# B&R Automation Studio project ACOPOStrak (part 2)

#### brdkEMModeToA.c - Converts an equipment module mode constant to a string representation.
```c
#include <brdkEM_func.h>

unsigned long brdkEMModeToA(signed long mode) {
	unsigned long pStr;
	switch(mode) {
		case MODE_UNDEFINED: 	pStr = (unsigned long)&"MODE_UNDEFINED"; 	break;	/* 0 */
		case MODE_PRODUCING: 	pStr = (unsigned long)&"MODE_PRODUCING"; 	break;	/* 1 */
		case MODE_MAINTENANCE: 	pStr = (unsigned long)&"MODE_MAINTENANCE"; 	break;	/* 2 */
		case MODE_MANUAL: 		pStr = (unsigned long)&"MODE_MANUAL"; 		break;	/* 3 */
		case MODE_CLEAN: 		pStr = (unsigned long)&"MODE_CLEAN"; 		break;	/* 16 */
		case MODE_JOG: 			pStr = (unsigned long)&"MODE_JOG"; 			break;	/* 17 */
		case MODE_CIP: 			pStr = (unsigned long)&"MODE_CIP"; 			break;	/* 18 */
		case MODE_CALIBRATING: 	pStr = (unsigned long)&"MODE_CALIBRATING"; 	break;	/* 19 */
		default: break;
	}
	return pStr;
}
```

#### brdkEM_func.c - Internal functions for brdkEM.
```c
#include <brdkEM_func.h>

static unsigned char semCreator = false;
SemCreate_typ SemCreateMUList;
char tmpStr[BRDK_MU_MAX_DESCRIPTION_STRING];

/* initialize the equipment module */
void brdkEMInitialize(brdkEM_typ* this, brdkEM_typ* parent) {
	int i;
	brdk_mu_setup_module_typ module;

	switch(this->internal.initSubstate) {

		case 0:
			if(this->setup.name[0] == 0) ST_name(0,(char*)&this->setup.name,(unsigned char)0); 														/* set module name to task name if not set*/
			brdkStrCpy((unsigned long)this->status.name,(unsigned long)this->setup.name);
			if(this->setup.status.stateSubstateMode) {
				brdkStrCpy((unsigned long)this->status.state,(unsigned long)brdkEMStateToA(this->state));
				brdkStrCpy((unsigned long)this->status.mode,brdkEMModeToA(this->mode));
			}
			if(this->setup.nameIdx > -1) brdkStrAppendUdintToA(this->setup.nameIdx,(unsigned long)&this->status.name, BRDK_STR_CONVERT_DECIMAL,-1);	/* add index to task name */
			this->internal.muList.parentIdx = -1;
			for(i=0; i<= BRDK_EM_MAX_CHILDREN; i++) this->internal.muList.childrenIdx[i] = -1;
			for(i=0; i<= BRDK_MU_MAX_SIBLINGS; i++) this->internal.muList.siblingIdx[i] = -1;
			if(!semCreator) {
				setSubStateText(this,(unsigned long)"creating global semaphore");
				semCreator = true;
				this->internal.initSubstate = 10;
			}
			else this->internal.initSubstate = 20;
			break;

		case 10:
			SemCreateMUList.enable = true;
			SemCreateMUList.initCount = 0;
			SemCreateMUList.maxCount = 1;
			SemCreate(&SemCreateMUList);
			if(SemCreateMUList.status != ERR_OK) setSubStateText(this,(unsigned long)"creating global semaphore");
			else {
				SemRelease(SemCreateMUList.ident);
				this->internal.muList.idx = addToMUList((unsigned long)this,0);
				if(this->internal.muList.idx != -1) {
					emListReady = true;
					this->internal.initSubstate = !this->setup.parent.name[0] ? 40 : 30;	/* check if the module has a parent name assigned */
				}
				else {
					setSubStateText(this,(unsigned long)"em list full. Expand BRDK_EM_MAX_EMS.");
					this->internal.initSubstate = 200;
				}
			}
			break;

		case 20:	/* add module to em list */
			if(!emListReady) setSubStateText(this,(unsigned long)"waiting for em list to be ready");
			else {
				brdkStrCpy((unsigned long)module.name,(unsigned long)this->setup.name);
				module.index = this->setup.nameIdx;
				this->internal.muList.idx = getMUIndex((unsigned long)this, &module);
				if(this->internal.muList.idx != -1) {
					if(moduleSleeping(this->internal.muList.idx)) {
						wakeMU(this->internal.muList.idx,(unsigned long)this);
						if(this->setup.status.last) {
							brdkStrMemMove((unsigned long)this->status.last[1],(unsigned long)this->status.last[0], sizeof(this->status.last[0])*BRDK_MU_MAX_LAST_SIZE);
							brdkStrCpy((unsigned long)this->status.last[0],(unsigned long)"module awake");
						}
						this->internal.initSubstate = 65000;
					}
					else {	/* module name already exists in the list */
						this->status.substate[0] = 0;	/* reset sub state text */
						if(this->setup.status.stateSubstateMode) {
							brdkStrCpy((unsigned long)tmpStr,(unsigned long)"module name ");
							brdkStrCat((unsigned long)tmpStr,(unsigned long)module.name);
							brdkStrCat((unsigned long)tmpStr,(unsigned long)" already used. Rename module.");
							setSubStateText(this,(unsigned long)tmpStr);
						}
						this->internal.muList.idx = -1;
						this->internal.initSubstate = 100;
					}
				}
				else {
					if(SemAcquire(SemCreateMUList.ident) != ERR_OK) setSubStateText(this,(unsigned long)"waiting global semaphore to be free");
					else {
						this->internal.muList.idx = addToMUList((unsigned long)this,0);
						SemRelease(SemCreateMUList.ident);
						setSubStateText(this,(unsigned long)"module added em list");
						if(this->internal.muList.idx != -1) this->internal.initSubstate = !this->setup.parent.name[0] ? 40 : 30;	/* check if the module has a parent name assigned */
						else {
							setSubStateText(this,(unsigned long)"em list full. Expand BRDK_EM_MAX_EMS.");
							this->internal.initSubstate = 200;
						}
					}
				}
			}
			break;

		case 30:	/* find parent */
			this->internal.muList.parentIdx = getMUIndex((unsigned long)this, &this->setup.parent);
			if(this->internal.muList.parentIdx == -1) setSubStateText(this,(unsigned long)"parent not found");
			else this->internal.initSubstate = 40;
			break;

		case 40:	/* find siblings */
			for(i=0; i<= BRDK_MU_MAX_SIBLINGS; i++) {
				if(this->setup.sibling[i].name[0] != 0) {
					this->internal.muList.siblingIdx[i] = getMUIndex((unsigned long)this, &this->setup.sibling[i]);
					if(this->internal.muList.siblingIdx[i] == -1) {
						if(this->setup.status.stateSubstateMode) {
							brdkStrCpy((unsigned long)tmpStr,(unsigned long)"sibling: ");
							brdkStrCat((unsigned long)tmpStr,(unsigned long)this->setup.sibling[i].name);
							brdkStrCat((unsigned long)tmpStr,(unsigned long)" not found");
							setSubStateText(this,(unsigned long)tmpStr);
						}
						break;
					}
				}
			}
			if(i>=BRDK_MU_MAX_SIBLINGS) {
				this->status.substate[0] = 0;	/* reset status text */
				this->internal.initSubstate = this->internal.SemCreate_0.ident == 0 ? 50 : 60;
			}
			break;

		case 50:
			this->internal.SemCreate_0.enable = true;
			this->internal.SemCreate_0.initCount = 0;
			this->internal.SemCreate_0.maxCount = 1;
			SemCreate(&this->internal.SemCreate_0);
			switch(this->internal.SemCreate_0.status) {

				case 0:	/* ERR_OK */
					SemRelease(this->internal.SemCreate_0.ident);		/* release the semaphore so it's ready */
					this->internal.initSubstate = 60;
					break;

				case 65535:	/* ERR_FUB_BUSY */
					break;

				default:
					setSubStateText(this,(unsigned long)"error creating the semaphore");
					break;

			}
			break;

		case 60:
			switch(this->setup.activation) {
				case BRDK_EM_ACTIVATE:
					this->internal.deactivateRequest = false;
					this->internal.initSubstate = 70;
					break;

				case BRDK_EM_ACTIVATE_BY_PARENT:
					if(parent != NULL) {
						if(!parent->internal.deactivateRequest) {
							this->internal.initSubstate = 70;
							this->internal.deactivateRequest = false;
						}
					}
					break;

				default: break;

			}
			break;

		case 70:
			setSubStateText(this,(unsigned long)"register child to parent");
			if(RegisterChild(this, parent) == 0) {
				this->internal.initSubstate = 65000;				/* add child to parent's children list */
				if(this->substate == 0) this->substate = 65000;		/* if substate is still 0 it's auto set to SC */
			}
			break;

		case 100: /* error module name already used. Check if anme is being changed */
			break;

	}
}

/* traverse and find the real interrupter */
unsigned long findInterrupter(unsigned long pEM) {
	if(((brdkEM_typ*)pEM)->internal.pInterrupter != pEM) return findInterrupter(((brdkEM_typ*)pEM)->internal.pInterrupter);
	return pEM;
}

/* flash functionality */
brdk_em_color_typ flashColor(brdkEM_typ* this, brdk_em_color_typ color) {
	if(this->internal.flashTime >= BRDK_EM_FLASH_TIME*2) this->internal.flashTime = 0;
	else this->internal.flashTime += this->status.cycleTime/1000;
	return this->internal.flashTime >= BRDK_EM_FLASH_TIME ? color : WHITE;
}

/* light tree functionality */
void lightTree(brdkEM_typ* this, brdk_em_color_typ color1, brdk_em_color_typ color2) {
	this->status.lightTree.red 		= color1 == RED || color2 == RED;
	this->status.lightTree.yellow 	= color1 == ORANGE || color2 == ORANGE;
	this->status.lightTree.blue 	= color1 == BLUE || color2 == BLUE;
	this->status.lightTree.green 	= color1 == GREEN || color2 == GREEN;
}

/* set default sub state text if not set in program */
void setSubStateText(brdkEM_typ* this, unsigned long pStr) {
	const int MAX_COUNTER = 99999;
	if(this->status.substate[0] == 0 && this->setup.status.stateSubstateMode) {
		if(pStr != 0) {
			brdkStrCpy((unsigned long)this->status.substate,pStr);
			this->internal.statusCnt.internalCounter = this->internal.statusCnt.internalCounter > MAX_COUNTER ? 0 : this->internal.statusCnt.internalCounter+1;		/* increase the status counter to indicate that a change was made */
		}
		else {
			if(this->description[0] == 0) {
				if(this->substate == 0) {
					brdkStrCpy((unsigned long)this->status.substate,(unsigned long)"0: waiting for state change (SC)");
					this->internal.statusCnt.internalCounter = this->internal.statusCnt.internalCounter > MAX_COUNTER ? 0 : this->internal.statusCnt.internalCounter+1;		/* increase the status counter to indicate that a change was made */
				}
				else if(this->internal.cmdSC) {
					switch(this->state) {
						case STATE_DEACTIVATED: brdkStrCpy((unsigned long)this->status.substate, (unsigned long)"SC: waiting for activate command"); break;
						case STATE_STOPPED: case STATE_COMPLETE: brdkStrCpy((unsigned long)this->status.substate, (unsigned long)"SC: waiting for reset command"); break;
						case STATE_IDLE: case STATE_SUSPENDED: case STATE_HELD:	brdkStrCpy((unsigned long)this->status.substate, (unsigned long)"SC: waiting for start command"); break;
						case STATE_ABORTED: brdkStrCpy((unsigned long)this->status.substate, (unsigned long)"SC: waiting for clear command"); break;
						default: brdkStrCpy((unsigned long)this->status.substate, (unsigned long)"SC: waiting for command"); break;
					}
					this->internal.statusCnt.internalCounter = this->internal.statusCnt.internalCounter > MAX_COUNTER ? 0 : this->internal.statusCnt.internalCounter+1;		/* increase the status counter to indicate that a change was made */
				}
			}
			else {
				brdkStrUdintToA(this->substate,(unsigned long)&this->status.substate,BRDK_STR_CONVERT_DECIMAL);
				brdkStrCat((unsigned long)this->status.substate, (unsigned long)": ");
				brdkStrCat((unsigned long)this->status.substate, (unsigned long)this->description);
				this->internal.statusCnt.internalCounter = this->internal.statusCnt.internalCounter > MAX_COUNTER ? 0 : this->internal.statusCnt.internalCounter+1;		/* increase the status counter to indicate that a change was made */
			}
		}
	}
}

/* if the parent mode is changed we also changes it for alle the children */
void setChildrenMode(brdkEM_typ* this) {
	int i;
	for(i=0; i <= BRDK_EM_MAX_CHILDREN; i++) {
		brdkEM_typ* child = getEm(this->internal.muList.childrenIdx[i]);
		if(child != NULL) {
			if(this->setup.reactTo == BRDK_EM_REACT_TO_NONE) child->mode = child->mode;
			else child->mode = this->mode;
		}
		else break;
	}
}

/* CHECKS IF ALL THE CHILDREN IS IN STATE */
void checkChildren(brdkEM_typ* this, brdk_em_states_typ STATE) {
	brdkEM_typ* parent;
	brdkEM_typ* child;
	if(this->internal.cmdSC) {
		int i = 0, j;
		while(i < this->status.childCount) {
			child = getEm(this->internal.muList.childrenIdx[i]);
			if(child != NULL) {
				j = i;
				if(child->state == STATE_ACTIVATING || child->state == STATE_DEACTIVATED || child->state == STATE_DEACTIVATING) i++;
				else {
					switch(child->setup.reactTo) {

						case BRDK_EM_REACT_TO_ALL:
							if(child->state == STATE) i++;
							break;

						case BRDK_EM_REACT_TO_ABORT_AND_STOP:
							if(STATE == STATE_ABORTED || STATE == STATE_STOPPED) {
								if(child->state == STATE) i++;
							}
							else i++;
							break;

						case BRDK_EM_REACT_TO_ABORT_ONLY:
							if(STATE == STATE_ABORTED) {
								if(child->state == STATE) i++;
							}
							else i++;
							break;

						case BRDK_EM_REACT_TO_STOP_ONLY:
							if(STATE == STATE_STOPPED) {
								if(child->state == STATE) i++;
							}
							else i++;
							break;

						case BRDK_EM_REACT_TO_NONE: case BRDK_EM_LISTEN_TO_ABORT_AND_STOP: case BRDK_EM_LISTEN_TO_ABORT_ONLY: case BRDK_EM_LISTEN_TO_STOP_ONLY:
							i++;
							break;

					}
				}
				if(j == i) {	/* index not increased */
					if(child->internal.waitingForIdx != -1) {	/* check to see if a child is also waiting for someone */
						if(this->internal.waitingForIdx != child->internal.waitingForIdx) { /* check if the index has changed - otherwise there is nothing to update in the name */
							if(this->setup.status.waitingFor) brdkStrCpy((unsigned long)this->status.waitingFor.name,(unsigned long)child->status.waitingFor.name);
							this->internal.waitingForIdx = child->internal.waitingForIdx;
						}
						if(this->internal.statusCnt.externalCounter != child->internal.statusCnt.externalCounter) {	/* check if there is a change in the status text */
							if(this->setup.status.waitingFor) brdkStrCpy((unsigned long)this->status.waitingFor.substate,(unsigned long)child->status.waitingFor.substate);
							this->internal.statusCnt.externalCounter = child->internal.statusCnt.externalCounter;
						}
					}
					else {
						if(this->internal.waitingForIdx != child->internal.muList.idx) { /* check if the index has changed - otherwise there is nothing to update in the name */
							if(this->setup.status.stateSubstateMode) {
								brdkStrCpy((unsigned long)this->status.waitingFor.name,(unsigned long)child->setup.name);
								brdkStrCpy((unsigned long)tmpStr, (unsigned long)"SC: waiting for ");
								brdkStrCat((unsigned long)tmpStr, (unsigned long)this->status.waitingFor.name);
								setSubStateText(this,(unsigned long)tmpStr);
							}
							this->internal.waitingForIdx = child->internal.muList.idx;
						}
						if(this->internal.statusCnt.externalCounter != child->internal.statusCnt.internalCounter) {	/* check if there is a change in the status text */
							if(this->setup.status.waitingFor) brdkStrCpy((unsigned long)this->status.waitingFor.substate,(unsigned long)child->status.substate);
							this->internal.statusCnt.externalCounter = child->internal.statusCnt.internalCounter;
						}
					}
					break;
				}
			}
			else break;
		}
		if(parentStateOK(this)) {
			if(i==this->status.childCount) {
				if(this->state == STATE_RESETTING || this->state == STATE_CLEARING) {	/* clear interrupted by data */
					brdkStrMemSet((unsigned long)&this->status.interruptedBy,0,sizeof(this->status.interruptedBy));
					this->internal.pInterrupter = 0;
				}
				if(this->internal.waitingForIdx != -1) {
					if(this->setup.status.waitingFor) brdkStrMemSet((unsigned long)&this->status.waitingFor,0,sizeof(this->status.waitingFor)); /* clear waiting for data */
					this->internal.waitingForIdx = -1;				/* reset waiting for index */
					this->internal.statusCnt.externalCounter = -1;	/* reset external status counter */
				}
				this->state = STATE;
			}
		}
		else {
			if(!this->status.waitingFor.name[0]) {
				parent = getEm(this->internal.muList.parentIdx);
				if(parent != NULL) {
					if(this->internal.waitingForIdx != parent->internal.muList.idx) { /* check if the index has changed - otherwise there is nothing to update */
						this->internal.waitingForIdx = parent->internal.muList.idx;
						if(parent->state == STATE_DEACTIVATED || parent->state == STATE_DEACTIVATING) setSubStateText(this,(unsigned long)"SC: parent is deactivated");
						else setSubStateText(this,(unsigned long)"SC: waiting for parent");
						if(this->setup.status.waitingFor) brdkStrCpy((unsigned long)this->status.waitingFor.name,(unsigned long)parent->setup.name);
					}
					if(this->internal.statusCnt.externalCounter != parent->internal.statusCnt.internalCounter) {	/* check if there is a change in the status text */
						if(this->setup.status.waitingFor) brdkStrCpy((unsigned long)this->status.waitingFor.substate,(unsigned long)parent->status.substate);
						this->internal.statusCnt.externalCounter = parent->internal.statusCnt.internalCounter;
					}
				}
			}
		}
	}
}

/* make sure eventual parent is also in same state before state change */
int parentStateOK(brdkEM_typ* this) {
	int status = false;
	brdkEM_typ* parent = getEm(this->internal.muList.parentIdx);
	if(parent != NULL) {
		switch(this->setup.reactTo) {
			case BRDK_EM_REACT_TO_ALL: 				status = (parent->state == this->state || this->internal.findParent); break;
			case BRDK_EM_REACT_TO_ABORT_AND_STOP: 	status = (this->state == STATE_ABORTING || this->state == STATE_STOPPING) ? (parent->state == this->state) : true; break;
			case BRDK_EM_REACT_TO_ABORT_ONLY:		status = (this->state == STATE_ABORTING) ? (parent->state == this->state) : true; break;
			case BRDK_EM_REACT_TO_STOP_ONLY:		status = (this->state == STATE_STOPPING) ? (parent->state == this->state) : true; break;
			case BRDK_EM_REACT_TO_NONE: case BRDK_EM_LISTEN_TO_ABORT_AND_STOP: case BRDK_EM_LISTEN_TO_ABORT_ONLY: case BRDK_EM_LISTEN_TO_STOP_ONLY:	status = true;
		}
	}
	else status = true;
	return status;
}

/* automatically take the module to it's parents state */
void findParent(brdkEM_typ* this, brdkEM_typ* parent, brdk_em_states_typ cmd, int numArgs, ...) {
	if(parent != NULL) {
		va_list list;
		int i;
		if(this->state == parent->state) this->internal.findParent = false;
		else {
			va_start(list, numArgs);
			for(i=0; i < numArgs; i++) {
				brdk_em_states_typ checkState = va_arg(list, brdk_em_states_typ);
				if(parent->state == checkState) {
					switch(cmd) {
						case STATE_RESETTING: this->cmd.reset = true; break;
						case STATE_STARTING: case STATE_UNHOLDING: case STATE_UNSUSPENDING: this->cmd.start = true; break;
						case STATE_EXECUTE:
							switch(checkState) {
								case STATE_HOLDING: case STATE_HELD: this->cmd.hold = true; break;
								case STATE_SUSPENDING: case STATE_SUSPENDED: this->cmd.suspend = true; break;
								case STATE_COMPLETING: case STATE_COMPLETE: this->cmd.complete = true; break;
								default: break;
							}
							break;
						default: break;
					}
				}
			}
		}
	}
}

/* observes if one of the children is in one of the states */
void observeChildrensState(brdkEM_typ* this, int numArgs, ...) {
	int i,j;
	brdkEM_typ* child;
	va_list list;																					/* define argument list variable */
	for(i=0; i <= BRDK_EM_MAX_CHILDREN; i++) {														/* check all children */
		child = getEm(this->internal.muList.childrenIdx[i]);
		if(child != NULL) {											/* */
			brdk_em_setup_react_typ reactTo = child->setup.reactTo;
			if(reactTo == BRDK_EM_REACT_TO_NONE || reactTo == BRDK_EM_REACT_TO_NONE || reactTo == BRDK_EM_LISTEN_TO_ABORT_AND_STOP || reactTo == BRDK_EM_LISTEN_TO_ABORT_ONLY || reactTo == BRDK_EM_LISTEN_TO_STOP_ONLY) this->state = this->state;
			else {
				va_start(list, numArgs);
				for(j=0; j < numArgs; j++) {
					brdk_em_states_typ child_state = va_arg(list, brdk_em_states_typ);
					if(child->state == child_state) {
						switch(child_state) {

							case STATE_ABORTING:
								if(reactTo == BRDK_EM_REACT_TO_ALL || reactTo == BRDK_EM_REACT_TO_ABORT_AND_STOP || reactTo == BRDK_EM_REACT_TO_ABORT_ONLY) {
									this->internal.pInterrupter = findInterrupter((unsigned long)child); /* save who went in aborted or aborting */
									this->state = STATE_ABORTING;
								}
								break;

							case STATE_STOPPING:
								if((this->internal.cmdSC || this->setup.skipStopSC) && (reactTo == BRDK_EM_REACT_TO_ALL || reactTo == BRDK_EM_REACT_TO_ABORT_AND_STOP || reactTo == BRDK_EM_REACT_TO_STOP_ONLY)) {
									this->internal.pInterrupter = findInterrupter((unsigned long)child); /* save who went in stopped or stopping */
									this->state = STATE_STOPPING;
								}
								break;

							case STATE_SUSPENDING:
								if(this->internal.cmdSC && reactTo == BRDK_EM_REACT_TO_ALL) {
									this->internal.pInterrupter = findInterrupter((unsigned long)child); /* save who went in suspending or suspended */
									this->state = STATE_SUSPENDING;
								}
								break;

							case STATE_HOLDING:
								if(this->internal.cmdSC && reactTo == BRDK_EM_REACT_TO_ALL) {
									this->internal.pInterrupter = findInterrupter((unsigned long)child); /* save who went in holding or held */
									this->state = STATE_HOLDING;
								}
								break;

							default:
								break;

						}
						va_end(list);
						break;
					}
				}
			}
		}
		else {
			va_end(list);
			break;
		}
	}
}

/* observes the parent state by the given states */
void observeParentState(brdkEM_typ* this, brdkEM_typ* parent, int numArgs, ...) {
	int i;
	brdk_em_setup_react_typ reactTo =  this->setup.reactTo;
	if(parent == NULL || reactTo == BRDK_EM_REACT_TO_NONE) this->state = this->state;
	else {
		va_list list;																									/* define argument list variable */
		va_start(list, numArgs);																						/* init list */
		for(i=0; i < numArgs; i++) if(parent->state==va_arg(list, brdk_em_states_typ)) {
			switch(parent->state) {

				case STATE_ABORTING:
					if(reactTo == BRDK_EM_REACT_TO_ALL || reactTo == BRDK_EM_REACT_TO_ABORT_AND_STOP || reactTo == BRDK_EM_REACT_TO_ABORT_ONLY || reactTo == BRDK_EM_LISTEN_TO_ABORT_AND_STOP || reactTo == BRDK_EM_LISTEN_TO_ABORT_ONLY) {
						this->state = parent->state; 	/* get next state item and check if it's equal to parent state. and then set chils state*/
						this->internal.pInterrupter = parent->internal.pInterrupter;
					}
					break;

				case STATE_STOPPING:
					if((this->internal.cmdSC || this->setup.skipStopSC) && (reactTo == BRDK_EM_REACT_TO_ALL || reactTo == BRDK_EM_REACT_TO_ABORT_AND_STOP || reactTo == BRDK_EM_REACT_TO_STOP_ONLY || reactTo == BRDK_EM_LISTEN_TO_STOP_ONLY)) {
						this->state = parent->state; 	/* get next state item and check if it's equal to parent state. and then set chils state*/
						this->internal.pInterrupter = parent->internal.pInterrupter;
					}
					break;

				case STATE_CLEARING:
					if(this->internal.cmdSC && (reactTo == BRDK_EM_REACT_TO_ALL || reactTo == BRDK_EM_REACT_TO_ABORT_AND_STOP || reactTo == BRDK_EM_REACT_TO_ABORT_ONLY)) this->state = parent->state; 	/* get next state item and check if it's equal to parent state. and then set chils state*/
					break;

				default:
					if(this->internal.cmdSC && reactTo == BRDK_EM_REACT_TO_ALL) this->state = parent->state; 	/* get next state item and check if it's equal to parent state. and then set chils state*/
					break;

			}
		}
		va_end(list);
	}																													/* cleanup the system stack */
}

/* check for commands -> STATE_STOPPING means check for command stop... */
void checkCommands(brdkEM_typ* this, brdkEM_typ* parent, int numArgs, ...) {
	brdkEM_typ* child;
	int i,j;
	if(this->internal.cmdSC || this->cmd.abort || (this->cmd.stop && this->setup.skipStopSC)) {
		va_list list;																											/* define argument list variable */
		va_start(list, numArgs);																								/* init list */
		for(i=0; i < numArgs; i++) {
			switch(va_arg(list, brdk_em_states_typ)) {

				case STATE_STOPPING:
					if(this->cmd.stop) {
						i = numArgs;
						this->internal.pInterrupter = (unsigned long)this; /* module interrupted itself */
						this->state = STATE_STOPPING;
					}
					break;

				case STATE_RESETTING:
					if(this->cmd.reset) {
						i = numArgs;
						this->state = STATE_RESETTING;
					}
					break;

				case STATE_CLEARING:
					if(this->cmd.clear) {
						this->state = STATE_CLEARING;
					}
					break;

				case STATE_STARTING:
					if(this->cmd.start) {
						i = numArgs;
						this->state = STATE_STARTING;
					}
					break;

				case STATE_HOLDING:
					if(this->cmd.hold) {
						i = numArgs;
						this->internal.pInterrupter = (unsigned long)this; /* module interrupted itself */
						this->state = STATE_HOLDING;
					}
					break;

				case STATE_UNHOLDING:
					if(this->cmd.start) {
						i = numArgs;
						this->state = STATE_UNHOLDING;
					}
					break;

				case STATE_SUSPENDING:
					if(this->cmd.suspend) {
						i = numArgs;
						this->internal.pInterrupter = (unsigned long)this; /* module interrupted itself */
						this->state = STATE_SUSPENDING;
					}
					break;

				case STATE_UNSUSPENDING:
					if(this->cmd.start) {
						i = numArgs;
						this->state = STATE_UNSUSPENDING;
					}
					break;

				case STATE_COMPLETING:
					if(this->cmd.complete) {
						i = numArgs;
						this->state = STATE_COMPLETING;
					}
					break;

				case STATE_ABORTING:
					if(this->cmd.abort) {
						i = numArgs;
						this->internal.pInterrupter = (unsigned long)this; /* module interrupted itself */
						this->state = STATE_ABORTING;
					}
					break;

				case STATE_ACTIVATING:
					/* wait for initialization complete */
					if(this->internal.initSubstate == 65000) {
						switch(this->setup.activation) {

							case BRDK_EM_ACTIVATE:
								this->state = STATE_ACTIVATING;
								break;

							case BRDK_EM_ACTIVATE_BY_PARENT:
								if(parent != NULL) {
									switch(parent->state) {
										case STATE_DEACTIVATING: case STATE_DEACTIVATED: setSubStateText(this,(unsigned long)"waiting for parent's activation"); break;
										default:
											if(!parent->internal.deactivateRequest) this->state = STATE_ACTIVATING;
											break;
									}
								}
								break;

							default:
								setSubStateText(this, (unsigned long)"waiting for activation");
								break;

						}
					}
					break;

				case STATE_DEACTIVATING:
					switch(this->setup.activation) {

						case BRDK_EM_DEACTIVATE:
							this->internal.deactivateRequest = true;
							for(j=0; j <= BRDK_EM_MAX_CHILDREN; j++) {		/* check all children */
								child = getEm(this->internal.muList.childrenIdx[j]);
								if(child != NULL) {
									if(child->state != STATE_DEACTIVATED && child->state && STATE_DEACTIVATING) break;
								}
							}
							if(j > BRDK_EM_MAX_CHILDREN) {
								i = numArgs;
								this->state = STATE_DEACTIVATING;
							}
							break;

						case BRDK_EM_ACTIVATE_BY_PARENT:
							if(parent != NULL) {
								switch(parent->state) {
									case STATE_DEACTIVATING: case STATE_DEACTIVATED: this->state = STATE_DEACTIVATING; break;

									case STATE_ABORTED: case STATE_STOPPED:
										/* check if parent has deactivation command and then follow */
										if(parent->internal.deactivateRequest) {
											this->internal.deactivateRequest = true;
											for(j=0; j <= BRDK_EM_MAX_CHILDREN; j++) {		/* check all children */
												child = getEm(this->internal.muList.childrenIdx[j]);
												if(child != NULL) {
													if(child->state != STATE_DEACTIVATED && child->state && STATE_DEACTIVATING) break;
												}
											}
											if(j > BRDK_EM_MAX_CHILDREN) {
												i = numArgs;
												this->state = STATE_DEACTIVATING;
											}
										}
										break;

									default: break;
								}
							}
							break;

						default:
							break;

					}
					break;

				default:
					break;

			}
		}
		va_end(list);
		/* check if an unvalid command has been given */
		this->status.unvalidatedCmd = this->state != this->internal.old.state ? false : this->cmd.abort || this->cmd.clear || this->cmd.stop || this->cmd.reset || this->cmd.start || this->cmd.hold || this->cmd.suspend || this->cmd.complete;
	}
}

/* Add's a child to the parents child list */
unsigned short RegisterChild(brdkEM_typ* this, brdkEM_typ* parent) {
	int i=0, j=0;
	if(parent != NULL) {
		for(i=0; i < BRDK_EM_MAX_CHILDREN; i++) {
			if(parent->internal.muList.childrenIdx[i] == this->internal.muList.idx) break;	/* child already exists in array. index is returned */
			else if(parent->internal.muList.childrenIdx[i] == -1) {							/* finds an empty spot in the array */
				j = SemAcquire(parent->internal.SemCreate_0.ident);							/* checks if the semaphore is free */
				if(j == ERR_OK) {
					parent->internal.muList.childrenIdx[i] = this->internal.muList.idx;		/* puts the index in the array */
					parent->status.childCount++;
					SemRelease(parent->internal.SemCreate_0.ident);							/* releases the semaphore again */
					i = ERR_OK;
				}
				else {
					i = j;	/* 33322: Semaphore with the specified ident does not exist   33323: Semaphore is being used */
					if(this->setup.status.stateSubstateMode) {
						brdkStrCpy((unsigned long)tmpStr,(unsigned long)"semaphore error: ");
						brdkStrAppendUdintToA(j,(unsigned long)tmpStr,10,-1);
						setSubStateText(this,(unsigned long)tmpStr);
					}
				}
				break;
			}
		}
		if(i == BRDK_EM_MAX_CHILDREN) {  /* error: child array too small. Solution: make child array bigger */
			setSubStateText(this,(unsigned long)"parent child array full. Increase BRDK_EM_MAX_CHILDREN.");
		}
	}
	return i;
}

/* Unregister a child */
unsigned short UnregisterChild(brdkEM_typ* this, brdkEM_typ* parent) {
	int i=65000,j;
	if(parent != NULL) {
		for(i=0; i < BRDK_EM_MAX_CHILDREN; i++) {
			if(parent->internal.muList.childrenIdx[i] == this->internal.muList.idx) {	/* child found */
				j = SemAcquire(parent->internal.SemCreate_0.ident);	/* checks if the semaphore is free */
				if(j == ERR_OK) {
					parent->internal.muList.childrenIdx[i] = -1;			/* pointer is removed from the array */
					parent->status.childCount--;
					for(j=i; j < BRDK_EM_MAX_CHILDREN; j++) parent->internal.muList.childrenIdx[j] = parent->internal.muList.childrenIdx[j+1];
					SemRelease(parent->internal.SemCreate_0.ident);		/* releases the semaphore again */
					i = ERR_OK;
					this->internal.muList.parentIdx = -1;
				}
				else {
					i = j;	/* 33322: Semaphore with the specified ident does not exist   33323: Semaphore is being used */
					if(this->setup.status.stateSubstateMode) {
						brdkStrCpy((unsigned long)tmpStr,(unsigned long)"semaphore error: ");
						brdkStrAppendUdintToA(j,(unsigned long)tmpStr,10,-1);
						setSubStateText(this,(unsigned long)tmpStr);
					}
				}
				break;
			}
		}
		if(i == BRDK_EM_MAX_CHILDREN) {  /* error: child not found in array */
			setSubStateText(this,(unsigned long)"child not found in parent array.");
		}
	}
	return i;
}
```

#### brdkMU_func.c - Internal functions for brdkMU.
```c
#include <brdkMU_func.h>

enum mu_state_typ
{
	MU_UNVALID,
	MU_ENABLED,
	MU_SLEEPING,
	MU_UPDATING
};

typedef struct brdk_mu_pointers_typ
{	enum mu_state_typ state;
	unsigned char type;	/* 0 = em, 1 = cm */
	unsigned long ptr;
} brdk_mu_pointers_typ;

static brdk_mu_pointers_typ muList[BRDK_MU_MAX_MODULES];
unsigned char emListReady = false;

/* addes a module mu list */
signed long addToMUList(unsigned long this, unsigned char type) {
	signed long i;
	for(i=0; i< BRDK_MU_MAX_MODULES; i++) {
		if(muList[i].ptr == this) return i;	/* module already inside list */
		else if(muList[i].ptr == 0) { 				/* find an empty slot in the list */
			muList[i].ptr = this;
			muList[i].state = MU_ENABLED;
			muList[i].type = type;
			return i;
		}
	}
	return -1;
}

/* returns the index in the em list of the wanted module */
signed long getMUIndex(unsigned long this, brdk_mu_setup_module_typ* module) {
	signed long i;
	brdkEM_typ* em;
	brdkCM_typ* cm;
	for(i=0; i < BRDK_MU_MAX_MODULES; i++) {
		if(muList[i].ptr != this) {
			if(muList[i].ptr != 0){
				if(muList[i].state != MU_UNVALID) {
					switch(muList[i].type) {
						case 0:
							em = (brdkEM_typ*)muList[i].ptr;
							if(!brdkStrCmp((unsigned long)em->setup.name,(unsigned long)module->name) && em->setup.nameIdx == module->index) return i;
							break;

						case 1:
							cm = (brdkCM_typ*)muList[i].ptr;
							if(!brdkStrCmp((unsigned long)cm->setup.name,(unsigned long)module->name) && cm->setup.nameIdx == module->index) return i;
							break;

					}
				}
			}
			else return -1; /* no further modules */
		}
	}
	return -1;
}

/* returns the pointer of the em */
brdkEM_typ* getEm(signed long idx) {
	if(idx != -1) {
		/* TODO - make check of unit type */
		if(muList[idx].state != MU_UNVALID && muList[idx].ptr != 0) return (brdkEM_typ*)muList[idx].ptr;
	}
	return NULL;
}

/* returns the pointer of the em */
brdkCM_typ* getCm(signed long idx) {
	if(idx != -1) {
		/* TODO - make check of unit type */
		if(muList[idx].state != MU_UNVALID && muList[idx].ptr != 0) return (brdkCM_typ*)muList[idx].ptr;
	}
	return NULL;
}

signed long sleepMU(signed long idx, unsigned long this) {
	if(idx != -1) {
		muList[idx].state = MU_UNVALID;
		switch(muList[idx].type) {
			case 0:
				TMP_alloc(sizeof(brdkEM_typ),(void*)&muList[idx].ptr);
				brdkStrMemCpy(muList[idx].ptr,this, sizeof(brdkEM_typ));
				break;

			case 1:
				TMP_alloc(sizeof(brdkCM_typ),(void*)&muList[idx].ptr);
				brdkStrMemCpy(muList[idx].ptr,this, sizeof(brdkCM_typ));
				break;

		}
		muList[idx].state = MU_SLEEPING;
		return idx;
	}
	return -1;
}

signed long wakeMU(signed long idx, unsigned long this) {
	if(idx != -1) {
		if(muList[idx].state == MU_SLEEPING) {
			muList[idx].state = MU_UNVALID;
			switch(muList[idx].type) {
				case 0:
					brdkStrMemCpy(this,muList[idx].ptr, sizeof(brdkEM_typ));	/* UPDATE THIS TO NAME BASE INSTEAD OF MEMORY */
					TMP_free(sizeof(brdkEM_typ),(void*)muList[idx].ptr);
					break;

				case 1:
					brdkStrMemCpy(this,muList[idx].ptr, sizeof(brdkCM_typ));	/* UPDATE THIS TO NAME BASE INSTEAD OF MEMORY */
					TMP_free(sizeof(brdkCM_typ),(void*)muList[idx].ptr);
					break;

			}
			muList[idx].state = MU_ENABLED;
		}
		muList[idx].state = MU_UNVALID;
		muList[idx].ptr = this;
		muList[idx].state = MU_ENABLED;
		return idx;
	}
	return -1;
}

/* returns if a module is sleeping or not */
unsigned char moduleSleeping(signed long idx) {
	return muList[idx].state == MU_SLEEPING;
}

/* updates the siblings state and sub state info for the em function block */
void updateSiblingInfo(signed long (*idxArr)[], brdk_mu_status_module_typ* status) {
	int i;
	brdkEM_typ* sibling;
	for(i=0; i<= BRDK_MU_MAX_SIBLINGS; i++) {
		sibling = getEm((*idxArr)[i]);
		if(sibling != NULL) {
			status[i].state = sibling->state;
			status[i].substate = sibling->substate;
			status[i].sleeping = sibling->status.sleeping;
			status[i].mode = sibling->mode;
		}
	}
}

/* gets the cycle time of the task the em structure is called inside */
unsigned long getCycleTime() {
	RTInfo_typ RTInfo_0;
	RTInfo_0.enable = 1;
	RTInfo(&RTInfo_0);
	return RTInfo_0.cycle_time;
}
```

- CHANGELOG - brdkMU change log file (not shown)

### Library Logical/Libraries/brdkSTR (ANSIC, version 1.04.0) - brdk string handling library. Expands string functionality.

#### brdkSTR.fun
```iecst
FUNCTION brdkStrAppendUdintToA : DINT (*Appends an UDINT to the end of a string. $RETURN=length;Length of the string.*) (*$GROUP=User,$CAT=User,$GROUPICON=User.png,$CATICON=User.png*)
	VAR_INPUT
		value : UDINT; (*UDINT value to be converted.*)
		pString : UDINT; (*String pointer to source string.*)
		base : USINT; (*0,10 = decimal, 2 = binary, 16 = hex.*)
		position : DINT; (*Append position. Negative numbers will count from end of string.*)
	END_VAR
END_FUNCTION

FUNCTION brdkStrAToDint : DINT (*Converts a string to a DINT type. $RETURN=value;DINT value.*) (*$GROUP=User,$CAT=User,$GROUPICON=User.png,$CATICON=User.png*)
	VAR_INPUT
		pString : UDINT; (*String pointer to source string.*)
		base : USINT; (*0,10 = decimal, 2 = binary, 16 = hex.*)
	END_VAR
END_FUNCTION

FUNCTION brdkStrAToUdint : UDINT (*Converts a string to an UDINT type. $RETURN=value;UDINT value.*) (*$GROUP=User,$CAT=User,$GROUPICON=User.png,$CATICON=User.png*)
	VAR_INPUT
		pString : UDINT; (*String pointer to source string.*)
		base : USINT; (*0,10 = decimal, 2 = binary, 16 = hex.*)
	END_VAR
END_FUNCTION

FUNCTION brdkStrCat : UDINT (*Appends a copy of the source string to the end of the destination string. $RETURN=address;Address after the string.*) (*$GROUP=User,$CAT=User,$GROUPICON=User.png,$CATICON=User.png*)
	VAR_INPUT
		pDestination : UDINT; (*Destination string pointer.*)
		pSource : UDINT; (*Source string pointer.*)
	END_VAR
END_FUNCTION

FUNCTION brdkStrCatAtChar : DINT (*Appends a copy of the source string to the char position of the destination string. $RETURN=index;Index in destination string where the source string is appended. -1 if char is not found.*) (*$GROUP=User,$CAT=User,$GROUPICON=User.png,$CATICON=User.png*)
	VAR_INPUT
		pDestination : UDINT; (*Destination string pointer.*)
		pSource : UDINT; (*Source string pointer.*)
		pChar : UDINT; (*Char pointer.*)
		direction : DINT; (*0 = first appearance of char, -1 = last appearance of char.*)
		greedy : BOOL; (*If true the source string is appended to the char position. If false the char is still present in the destination string.*)
	END_VAR
END_FUNCTION

FUNCTION brdkStrCharAt : USINT (*Returns the character at the specified index. $RETURN=coding;ASCII coding of the char.*) (*$GROUP=User,$CAT=User,$GROUPICON=User.png,$CATICON=User.png*)
	VAR_INPUT
		pString : UDINT; (*String pointer to source string.*)
		index : UDINT; (*Look up index.*)
		pChar : UDINT; (*Char pointer to char to look up.*)
	END_VAR
END_FUNCTION

FUNCTION brdkStrCharCount : DINT (*Finds how many times a character appears in a string. $RETURN=count;Char count. -1 if error.*) (*$GROUP=User,$CAT=User,$GROUPICON=User.png,$CATICON=User.png*)
	VAR_INPUT
		pString : UDINT; (*String pointer to source string.*)
		pChar : UDINT; (*Pointer to search char.*)
	END_VAR
END_FUNCTION

FUNCTION brdkStrCmp : DINT (*Compares character(s) from string1 to string2. $RETURN=result;0 means that the two string are equal.*)
	VAR_INPUT
		pString1 : UDINT; (*String1 pointer.*)
		pString2 : UDINT; (*String2 pointer.*)
	END_VAR
END_FUNCTION

FUNCTION brdkStrCpy : UDINT (*Copies a string to another string. $RETURN=address;Address after the string.*) (*$GROUP=User,$CAT=User,$GROUPICON=User.png,$CATICON=User.png*)
	VAR_INPUT
		pDestination : UDINT; (*Destination string pointer.*)
		pSource : UDINT; (*Source string pointer.*)
	END_VAR
END_FUNCTION

FUNCTION brdkStrCrc32 : UDINT (*Calculates a CRC32 checksum based on the input string. $RETURN=checksum;Checksum of the string.*) (*$GROUP=User,$CAT=User,$GROUPICON=User.png,$CATICON=User.png*)
	VAR_INPUT
		pString : UDINT; (*String pointer.*)
	END_VAR
END_FUNCTION

FUNCTION brdkStrDintToA : DINT (*Converts a DINT into a STRING type. $RETURN=length;Length of the string.*) (*$GROUP=User,$CAT=User,$GROUPICON=User.png,$CATICON=User.png*)
	VAR_INPUT
		value : DINT; (*DINT value to be converted.*)
		pString : UDINT; (*String pointer to source string.*)
		base : USINT; (*0,10 = decimal, 2 = binary, 16 = hex.*)
	END_VAR
END_FUNCTION

FUNCTION brdkStrEncode : DINT (*Encodes a string into different formats. $RETURN=address;Address after the string.*) (*$GROUP=User,$CAT=User,$GROUPICON=User.png,$CATICON=User.png*)
	VAR_INPUT
		pDestination : UDINT; (*Destination string pointer.*)
		pSource : UDINT; (*Source string pointer.*)
		format : USINT; (*0 = UTF-8*)
	END_VAR
END_FUNCTION

FUNCTION brdkStrFill : DINT (*Inserts amount of character(s) to the specified position of the string. $RETURN=length;Length of the string. -1 if error.*) (*$GROUP=User,$CAT=User,$GROUPICON=User.png,$CATICON=User.png*)
	VAR_INPUT
		pString : UDINT; (*String pointer to source string.*)
		amount : DINT; (*Fill char amount.*)
		pChar : UDINT; (*Fill char. If 0 whitespace is used.*)
		position : DINT; (*Fill position. Negative numbers will count from end of string.*)
	END_VAR
END_FUNCTION

FUNCTION brdkStrIndexOf : DINT (*Returns the index within this string of the first or last occurrence of the specified character. $RETURN=index;Index of the char. -1 if char is not found.*) (*$GROUP=User,$CAT=User,$GROUPICON=User.png,$CATICON=User.png*)
	VAR_INPUT
		pString : UDINT; (*String pointer to source string.*)
		pChar : UDINT; (*Char pointer to char to look up.*)
		direction : DINT; (*0 = search from left, -1 = search from right.*)
	END_VAR
END_FUNCTION

FUNCTION brdkStrInsertAtPos : DINT (*Inserts a string into another string at a specified position. $RETURN=length;Length of the string. -1 if error.*) (*$GROUP=User,$CAT=User,$GROUPICON=User.png,$CATICON=User.png*)
	VAR_INPUT
		pString : UDINT; (*String pointer to source string.*)
		pInsert : UDINT; (*String pointer to insert string.*)
		position : DINT; (*Insert position. Negative numbers will count from end of string.*)
	END_VAR
END_FUNCTION

FUNCTION brdkStrIsEmpty : BOOL (*Returns false or true depending of characters are present in the first position of the string. $RETURN=false/true;Position [0] = /0 = false. Position [0] != /0 = true.*) (*$GROUP=User,$CAT=User,$GROUPICON=User.png,$CATICON=User.png*)
	VAR_INPUT
		pString : UDINT; (*String pointer.*)
	END_VAR
END_FUNCTION

FUNCTION brdkStrLen : DINT (*Returns the number of characters in a string. Stops at \0. $RETURN=length;length of the string*) (*$GROUP=User,$CAT=User,$GROUPICON=User.png,$CATICON=User.png*)
	VAR_INPUT
		pString : UDINT; (*String pointer.*)
	END_VAR
END_FUNCTION

FUNCTION brdkStrMemCmp : DINT (*Compares amount of character(s) from area1 to area2. $RETURN=result;0 means that the two areas are equal.*) (*$GROUP=User,$CAT=User,$GROUPICON=User.png,$CATICON=User.png*)
	VAR_INPUT
		pArea1 : UDINT; (*Area1 pointer.*)
		pArea2 : UDINT; (*Area2 pointer.*)
		amount : UDINT; (*Amount of character(s) to be comared.*)
	END_VAR
END_FUNCTION

FUNCTION brdkStrMemCpy : UDINT (*Copies amount of character(s) from source to destination. $RETURN=address;Address after the destination.*) (*$GROUP=User,$CAT=User,$GROUPICON=User.png,$CATICON=User.png*)
	VAR_INPUT
		pDestination : UDINT; (*Destination pointer.*)
		pSource : UDINT; (*Source pointer.*)
		amount : UDINT; (*Amount of character(s) to be copied.*)
	END_VAR
END_FUNCTION

FUNCTION brdkStrMemMove : UDINT (*Moves amount of character(s) from source to destination. $RETURN=address;Address after the destination.*) (*$GROUP=User,$CAT=User,$GROUPICON=User.png,$CATICON=User.png*)
	VAR_INPUT
		pDestination : UDINT; (*Destination pointer.*)
		pSource : UDINT; (*Source pointer.*)
		amount : UDINT; (*Amount of character(s) to be moved.*)
	END_VAR
END_FUNCTION

FUNCTION brdkStrMemSet : UDINT (*Fills amount of character(s) to destination. $RETURN=address;Address after the destination.*) (*$GROUP=User,$CAT=User,$GROUPICON=User.png,$CATICON=User.png*)
	VAR_INPUT
		pDestination : UDINT; (*Destination pointer.*)
		value : USINT; (*Initialization value.*)
		amount : UDINT; (*Amount of character(s) to be initialized.*)
	END_VAR
END_FUNCTION

FUNCTION brdkStrMove : UDINT (*Moves a string to another string. $RETURN=address;Address after the string.*) (*$GROUP=User,$CAT=User,$GROUPICON=User.png,$CATICON=User.png*)
	VAR_INPUT
		pDestination : UDINT; (*Destination string pointer.*)
		pSource : UDINT; (*Source string pointer.*)
	END_VAR
END_FUNCTION

FUNCTION brdkStrNCpy : UDINT (*Copies a string to another string. If the function encounters a null character in the source string, the function will add null characters to the destination string until amount character(s) have been written. $RETURN=address;Address after the string.*) (*$GROUP=User,$CAT=User,$GROUPICON=User.png,$CATICON=User.png*)
	VAR_INPUT
		pDestination : UDINT; (*Destination string pointer.*)
		pSource : UDINT; (*Source string pointer.*)
		amount : UDINT; (*Amount of character(s) to be moved.*)
	END_VAR
END_FUNCTION

FUNCTION brdkStrRemove : UDINT (*Removes character(s) from a string from a specified position. $RETURN=address;Address after the string.*) (*$GROUP=User,$CAT=User,$GROUPICON=User.png,$CATICON=User.png*)
	VAR_INPUT
		pString : UDINT; (*Source string pointer.*)
		start : DINT; (*Index of where to start in the string. Negative numbers start from the end of the string.*)
		length : DINT; (*0 means to the end of the string. Negative length is subtracted from the end of the string. Is start is negative length is subtracted from the start of the string. *)
	END_VAR
END_FUNCTION

FUNCTION brdkStrRepeat : DINT (*Repeats a string a specified number of times. $RETURN=length;Length of the string.*) (*$GROUP=User,$CAT=User,$GROUPICON=User.png,$CATICON=User.png*)
	VAR_INPUT
		pString : UDINT; (*String pointer to source string.*)
		times : DINT; (*Number of times the string should be repeated.*)
	END_VAR
END_FUNCTION

FUNCTION brdkStrReplace : DINT (*Replaces some characters with some other characters in a string. $RETURN=number;Number of replacements done.*) (*$GROUP=User,$CAT=User,$GROUPICON=User.png,$CATICON=User.png*)
	VAR_INPUT
		pString : UDINT; (*String pointer to source string.*)
		pFind : UDINT; (*String pointer to find string.*)
		pReplace : UDINT; (*String pointer to replacement string:*)
	END_VAR
END_FUNCTION

FUNCTION brdkStrReverse : DINT (*Reverses a string from start position to end position. $RETURN=count;Number of reverses done. -1 if error.*) (*$GROUP=User,$CAT=User,$GROUPICON=User.png,$CATICON=User.png*)
	VAR_INPUT
		pString : UDINT; (*String pointer to source string.*)
		startPosition : DINT; (*Start position. Must be a positive number and less than length.*)
		endPosition : DINT; (*End position. Must be less than length unless it's a negative numbers which will count from end of string.*)
	END_VAR
END_FUNCTION

FUNCTION brdkStrReverseWords : DINT (*Reverses words in a string. $RETURN=count;Number of words reversed.*) (*$GROUP=User,$CAT=User,$GROUPICON=User.png,$CATICON=User.png*)
	VAR_INPUT
		pString : UDINT; (*String pointer to source string.*)
	END_VAR
END_FUNCTION

FUNCTION brdkStrSearch : DINT (*Searches a string for a specified string. $RETURN=position; Position of the match. -1 if no match.*) (*$GROUP=User,$CAT=User,$GROUPICON=User.png,$CATICON=User.png*)
	VAR_INPUT
		pString : UDINT; (*String pointer to source string.*)
		pSearchString : UDINT; (*String pointer to search string.*)
	END_VAR
END_FUNCTION

FUNCTION brdkStrSlice : DINT (*Slices a part of a string. $RETURN=length;Length of the string. -1 if error.*) (*$GROUP=User,$CAT=User,$GROUPICON=User.png,$CATICON=User.png*)
	VAR_INPUT
		pString : UDINT; (*String pointer to source string.*)
		start : DINT; (*Start position.*)
		end : DINT; (*End position.*)
	END_VAR
END_FUNCTION

FUNCTION brdkStrSubStr : DINT (*Returns a part of a string. $RETURN=length;Length of the destination string. -1 if error.*) (*$GROUP=User,$CAT=User,$GROUPICON=User.png,$CATICON=User.png*)
	VAR_INPUT
		pDestination : UDINT; (*Destination string pointer.*)
		pSource : UDINT; (*Source string pointer.*)
		start : DINT; (*Index of where to start in the string. Negative numbers start from the end of the string.*)
		length : DINT; (*0 means to the end of the string. Negative length is subtracted from the end of the string. Is start is negative length is subtracted from the start of the string. *)
	END_VAR
END_FUNCTION

FUNCTION brdkStrToDec : DINT (*Converts a string of hexadecimal values to ASCII characters. $RETURN=length;Length of the string. -1 if error.*) (*$GROUP=User,$CAT=User,$GROUPICON=User.png,$CATICON=User.png*)
	VAR_INPUT
		pString : UDINT; (*String pointer to source string.*)
	END_VAR
END_FUNCTION

FUNCTION brdkStrToHex : DINT (*Converts a string of ASCII characters to hexadecimal values. $RETURN=length;Length of the string.*) (*$GROUP=User,$CAT=User,$GROUPICON=User.png,$CATICON=User.png*)
	VAR_INPUT
		pString : UDINT; (*String pointer to source string.*)
	END_VAR
END_FUNCTION

FUNCTION brdkStrToLowerCase : DINT (*Converts a string to lowercase letters. $RETURN=number;Number of characters changed.*) (*$GROUP=User,$CAT=User,$GROUPICON=User.png,$CATICON=User.png*)
	VAR_INPUT
		pString : UDINT; (*String pointer to source string.*)
	END_VAR
END_FUNCTION

FUNCTION brdkStrToUpperCase : DINT (*Converts a string to uppercase letters. $RETURN=number;Number of characters changed.*) (*$GROUP=User,$CAT=User,$GROUPICON=User.png,$CATICON=User.png*)
	VAR_INPUT
		pString : UDINT; (*String pointer to source string.*)
	END_VAR
END_FUNCTION

FUNCTION brdkStrToUpperCaseWords : DINT (*Convert the first character of each word to uppercase. (title()). $RETURN=number;Number of characters changed.*) (*$GROUP=User,$CAT=User,$GROUPICON=User.png,$CATICON=User.png*)
	VAR_INPUT
		pString : UDINT; (*String pointer to source string.*)
	END_VAR
END_FUNCTION

FUNCTION brdkStrTrim : DINT (*Removes whitespaces from a string. $RETURN=number;Number of whitespaces removed from string.*) (*$GROUP=User,$CAT=User,$GROUPICON=User.png,$CATICON=User.png*)
	VAR_INPUT
		pString : UDINT; (*String pointer to source string.*)
		direction : DINT; (*0 = both sides, 1 = left side only, -1 = right side only.*)
	END_VAR
END_FUNCTION

FUNCTION brdkStrUdintToA : DINT (*Converts an UDINT into a STRING type. $RETURN=length;Length of the string.*) (*$GROUP=User,$CAT=User,$GROUPICON=User.png,$CATICON=User.png*)
	VAR_INPUT
		value : UDINT; (*UDINT value to be converted.*)
		pString : UDINT; (*String pointer to source string.*)
		base : USINT; (*0,10 = decimal, 2 = binary, 16 = hex.*)
	END_VAR
END_FUNCTION
```

- CHANGELOG - brdkSTR change log (not shown)

### Program Logical/Modules/Main/Main (IEC)

#### Types.typ
```iecst
TYPE
	local_typ : 	STRUCT
		shuttleCount : USINT; (*nr of shuttles added*)
		shuttleFub : ARRAY[0..MAX_NUM_SHUTTLES]OF shuttleFub_typ;
	END_STRUCT;
	shuttleFub_typ : 	STRUCT
		MC_Stop_0 : MC_Stop; (*Function block for stopping shuttles*)
	END_STRUCT;
END_TYPE
```

#### Variables.var
```iecst
VAR
	em : brdkEM; (*Equipment module*)
END_VAR
VAR CONSTANT
	MAX_NUM_SHUTTLES : USINT := 49; (*Maximum Shuttles Handled by the Trak (+1)*)
END_VAR
(*sequence control*)
VAR
	ShuttleAxis : ARRAY[0..MAX_NUM_SHUTTLES] OF McAxisType;
	i : USINT;
END_VAR
(*FUB*)
VAR
	MC_BR_AsmPowerOn_AcpTrak_0 : MC_BR_AsmPowerOn_AcpTrak;
	MC_BR_AsmPowerOff_AcpTrak_0 : MC_BR_AsmPowerOff_AcpTrak;
	MC_BR_AsmGetShuttle_AcpTrak_0 : MC_BR_AsmGetShuttle_AcpTrak;
	this : local_typ;
	MC_BR_AsmReadStatus_AcpTrak_0 : MC_BR_AsmReadStatus_AcpTrak;
	MC_BR_AsmReset_AcpTrak_0 : MC_BR_AsmReset_AcpTrak;
	MC_BR_AsmReadInfo_AcpTrak_0 : MC_BR_AsmReadInfo_AcpTrak;
	SizeofUserdata : UDINT;
	idx : USINT;
	MC_BR_AsmDeleteShuttle_AcpTrak_0 : MC_BR_AsmDeleteShuttle_AcpTrak;
END_VAR
```

#### Main.st
```iecst
PROGRAM _INIT

    (* Write this value into the Size of Userdata in the Shuttle Stereotype configuration *)
    SizeofUserdata := SIZEOF(gShuttleUserData);

	//dummy call
	gTrack1;
	gTrack2;
	gTrack3;
	gTrack4;
	gTrack5;
	gTrack6;

    gMain.status.simulation := DiagCpuIsSimulated();
	IF gMain.status.simulation THEN
		gMain.cmd.reset := TRUE;
	END_IF

END_PROGRAM

PROGRAM _CYCLIC

	IF gMain.status.error THEN
		em.cmd.abort := TRUE;
	END_IF

	CASE em.mode OF

		MODE_PRODUCING:	// #1
			CASE em.state OF

				STATE_STOPPED:

					CASE em.substate OF
						0:
							em.description := 'waiting for communication to segments is ok';
							IF gMain.status.communication THEN
								em.substate := 10;
							END_IF
						10:
							em.description := 'waiting for assembly ready signal - estop ok?';
							IF gMain.status.ready OR gMain.status.power THEN
								em.substate := 20;
							ELSIF NOT gMain.status.communication THEN
								em.substate := 0;
							END_IF
						20:
							em.description := 'track ready, waiting for reset cmd';
							IF gMain.cmd.reset THEN
								gMain.cmd.reset := FALSE;
								idx := this.shuttleCount := 0;
								em.cmd.reset	:= TRUE;
								em.cmd.sc 		:= TRUE;
							ELSIF NOT gMain.status.ready OR NOT gMain.status.communication THEN
								gMain.cmd.reset := FALSE;
								em.cmd.sc 		:= FALSE;
								em.substate := 0;
							END_IF
					END_CASE

				STATE_RESETTING:

					CASE em.substate OF
						0:
							em.description := 'power on';
							IF MC_BR_AsmReadStatus_AcpTrak_0.AssemblyReady AND MC_BR_AsmReadStatus_AcpTrak_0.Valid THEN
								MC_BR_AsmPowerOn_AcpTrak_0.Execute 	:= FALSE;
								em.substate							:= 10;
							ELSE
								MC_BR_AsmPowerOn_AcpTrak_0.Execute := TRUE;
							END_IF
						10:
							em.description := 'check for shuttles on this sector';
							MC_BR_AsmGetShuttle_AcpTrak_0.Enable := TRUE;
							IF MC_BR_AsmGetShuttle_AcpTrak_0.Valid THEN
								idx := 0;
								em.substate := 20;
							END_IF
						20:
							em.description := 'loop through shuttles and save it';
							MC_BR_AsmGetShuttle_AcpTrak_0.Next := FALSE;
							IF MC_BR_AsmGetShuttle_AcpTrak_0.TotalCount > 0 THEN
								ShuttleAxis[idx] := MC_BR_AsmGetShuttle_AcpTrak_0.Axis;
								em.substate := 30;
							END_IF
						30:
							em.description := 'get next shuttle or move on';
							IF MC_BR_AsmGetShuttle_AcpTrak_0.RemainingCount > 0 THEN
								MC_BR_AsmGetShuttle_AcpTrak_0.Next := TRUE;
								idx := idx + 1;
								em.substate := 20;
							ELSE
								em.substate := SC;
							END_IF
						SC://state complete
							em.description := 'waiting for childs';
							this.shuttleCount := idx;
							idx := 0;
							MC_BR_AsmGetShuttle_AcpTrak_0.Enable := FALSE;
							em.cmd.sc := TRUE;
					END_CASE

				STATE_IDLE:
					em.description := 'Wait for start command';
					IF gMain.cmd.start THEN
						gMain.cmd.start := FALSE;
						em.cmd.start	:= TRUE;
						em.cmd.sc		:= TRUE;
					END_IF

				STATE_STARTING:
					em.cmd.sc := TRUE;
					em.description := 'waiting for children';

				STATE_EXECUTE:
					em.description := 'Waiting for stop command';
					IF gMain.cmd.stop THEN
						gMain.cmd.stop 	:= FALSE;
						em.cmd.stop 	:= TRUE;
					END_IF
					em.cmd.sc := TRUE;

				STATE_STOPPING:
					em.description := 'Stop all shuttles - normal';
					FOR i := 0 TO MAX_NUM_SHUTTLES DO
						this.shuttleFub[i].MC_Stop_0.Deceleration := 10.0;
						this.shuttleFub[i].MC_Stop_0.Execute := TRUE;
					END_FOR
					em.cmd.sc := TRUE;

				STATE_ABORTING:
					em.description := 'Stop all shuttles - fast';
					FOR i := 0 TO MAX_NUM_SHUTTLES DO
						this.shuttleFub[i].MC_Stop_0.Deceleration := 35.0;
						this.shuttleFub[i].MC_Stop_0.Execute := TRUE;
					END_FOR
					em.cmd.sc := TRUE;

				STATE_ABORTED:
					em.description := 'assembly fault';
					IF gMain.cmd.clear THEN
						gMain.cmd.clear := FALSE;
						em.cmd.clear := TRUE;
					END_IF

				STATE_CLEARING:
					CASE em.substate OF
						0:
							em.description := 'delete all shuttles';
							MC_BR_AsmDeleteShuttle_AcpTrak_0.Execute := TRUE;
							MC_BR_AsmDeleteShuttle_AcpTrak_0.Command :=  mcACPTRAK_SH_DELETE_ALL;
							em.substate := 10;

						10:
							em.description := 'waiting for delete all shuttles done';
							IF MC_BR_AsmDeleteShuttle_AcpTrak_0.Done THEN
								MC_BR_AsmDeleteShuttle_AcpTrak_0.Execute := FALSE;
								em.substate := 20;
							END_IF

						20:
							em.description := 'reset error';
							brsmemset(ADR(ShuttleAxis),0,SIZEOF(ShuttleAxis));
							MC_BR_AsmReset_AcpTrak_0.Execute := TRUE;
							em.substate := 30;

						30:
							em.description := 'waiting for error reset done';
							IF MC_BR_AsmReset_AcpTrak_0.Done OR NOT gMain.status.error THEN
								MC_BR_AsmReset_AcpTrak_0.Execute := FALSE;
								em.cmd.sc := TRUE;
							END_IF
					END_CASE

				ELSE	// if need add the missing states
					em.cmd.sc := TRUE;

			END_CASE

		MODE_MANUAL: // #3
			CASE em.state OF

				STATE_STOPPED:
					em.description := 'this is a good place to write what the module is waiting for';

				STATE_RESETTING:

				STATE_IDLE:

				STATE_STARTING:

				STATE_EXECUTE:

				STATE_STOPPING:

				ELSE	// if need add the missing states
					em.cmd.sc := TRUE;

			END_CASE

		ELSE
			em.cmd.sc := TRUE;

	END_CASE

	FOR i := 0 TO MAX_NUM_SHUTTLES DO
		IF ShuttleAxis[i].controlif <> 0 THEN
			this.shuttleFub[i].MC_Stop_0.Axis			:= ADR(ShuttleAxis[i]);
			this.shuttleFub[i].MC_Stop_0.Deceleration	:= 2.0;
			this.shuttleFub[i].MC_Stop_0();
			IF this.shuttleFub[i].MC_Stop_0.Done THEN
				this.shuttleFub[i].MC_Stop_0.Execute := FALSE;
			END_IF
		ELSE
			this.shuttleFub[i].MC_Stop_0.Execute := FALSE;
		END_IF
	END_FOR

	MC_BR_AsmPowerOn_AcpTrak_0.Assembly := ADR(gAssembly_1);
	MC_BR_AsmPowerOn_AcpTrak_0();

	MC_BR_AsmPowerOff_AcpTrak_0.Assembly := ADR(gAssembly_1);
	MC_BR_AsmPowerOff_AcpTrak_0();

	MC_BR_AsmReadStatus_AcpTrak_0.Assembly 	:= ADR(gAssembly_1);
	MC_BR_AsmReadStatus_AcpTrak_0.Enable	:= TRUE;
	MC_BR_AsmReadStatus_AcpTrak_0();

	MC_BR_AsmGetShuttle_AcpTrak_0.Assembly	:= ADR(gAssembly_1);
	MC_BR_AsmGetShuttle_AcpTrak_0();

	MC_BR_AsmReadInfo_AcpTrak_0.Assembly := ADR(gAssembly_1);
	MC_BR_AsmReadInfo_AcpTrak_0.Enable := TRUE;
	MC_BR_AsmReadInfo_AcpTrak_0();

	MC_BR_AsmReset_AcpTrak_0.Assembly := ADR(gAssembly_1);
	MC_BR_AsmReset_AcpTrak_0();

	MC_BR_AsmDeleteShuttle_AcpTrak_0.Assembly := ADR(gAssembly_1);
	MC_BR_AsmDeleteShuttle_AcpTrak_0();

	em();								// call the module

	gMain.status.ready := MC_BR_AsmReadInfo_AcpTrak_0.AssemblyInfo.ReadyForPowerOn AND MC_BR_AsmReadInfo_AcpTrak_0.Valid;
	gMain.status.power := MC_BR_AsmReadStatus_AcpTrak_0.AssemblyReady AND MC_BR_AsmReadStatus_AcpTrak_0.Valid;
	gMain.status.communication := MC_BR_AsmReadInfo_AcpTrak_0.AssemblyInfo.CommunicationReady AND MC_BR_AsmReadInfo_AcpTrak_0.Valid;
	gMain.status.error := MC_BR_AsmReadStatus_AcpTrak_0.AssemblyErrorStop AND MC_BR_AsmReadStatus_AcpTrak_0.Valid;

END_PROGRAM

PROGRAM _EXIT
	(* Insert code here *)

END_PROGRAM
```

### MainGlobal.typ - Global data types
```iecst
TYPE
	main_interface_typ : 	STRUCT
		cmd : main_if_cmd_typ;
		status : main_if_status_typ;
	END_STRUCT;
	main_if_cmd_typ : 	STRUCT
		reset : BOOL; (*Power on assembly*)
		start : BOOL; (*Start all shuttles*)
		stop : BOOL; (*Stop all shuttles*)
		clear : BOOL; (*Clear assembly error*)
		safety : main_if_cmd_safety_typ; (*safety*)
	END_STRUCT;
	main_if_cmd_safety_typ : 	STRUCT
		reset : BOOL; (*reset safety*)
	END_STRUCT;
	main_if_status_typ : 	STRUCT
		power : BOOL; (*power on*)
		ready : BOOL; (*ready to power on*)
		error : BOOL; (*assembly fault*)
		simulation : BOOL; (*target is simulated*)
		communication : BOOL; (*communication to all segments ok*)
		safety : main_if_status_safety_typ; (*safety*)
	END_STRUCT;
	main_if_status_safety_typ : 	STRUCT
		moduleOK : BOOL; (*communication ok*)
		ready : BOOL; (*safety ready*)
		resetNeeded : BOOL; (*safety reset needed*)
		started : BOOL; (*safety running*)
	END_STRUCT;
END_TYPE
```

### MainGlobal.var - Global variables
```iecst
VAR
	gMain : main_interface_typ;
END_VAR
```

### Program Logical/Modules/Sectors/Track1Sector/Track1Sector (IEC) - Task for handling Track 2 sectors

#### Main.st - Init, cyclic, exit code
```iecst
PROGRAM _INIT

	MC_BR_TrgPointEnable_AcpTrak_0.Enable := TRUE;
	MC_BR_BarrierCommand_AcpTrak_0.Command := mcACPTRAK_BARRIER_ADD_TICKETS;
	MC_BR_BarrierCommand_AcpTrak_0.AdvancedParameters.TicketCount := 1;

	myTestDirection := mcDIR_POSITIVE;

END_PROGRAM

PROGRAM _CYCLIC

	em.setup.parent.name := 'Main';

	setup;

	CASE em.state OF
		STATE_STOPPED:
			idx := 0;
			MC_BR_SecGetShuttle_AcpTrak_0.Enable := FALSE;
			em.cmd.sc := TRUE;

		STATE_RESETTING:
			CASE em.substate OF
				0:
					em.description := 'check for shuttles on this sector';
					MC_BR_SecGetShuttle_AcpTrak_0.Enable := gMain.status.power;
					IF MC_BR_SecGetShuttle_AcpTrak_0.Valid THEN
						em.substate := 10;
					END_IF
				10:
					em.description := 'loop through shuttles and save it';
					MC_BR_SecGetShuttle_AcpTrak_0.Next := FALSE;
					IF MC_BR_SecGetShuttle_AcpTrak_0.TotalCount > 0 THEN
						this.axis[idx] := MC_BR_SecGetShuttle_AcpTrak_0.Axis;
						em.substate := 20;
					ELSE
						em.cmd.sc := TRUE; //no shuttles
					END_IF
				20:
					em.description := 'get next shuttle or move on';
					IF MC_BR_SecGetShuttle_AcpTrak_0.RemainingCount > 0 THEN
						MC_BR_SecGetShuttle_AcpTrak_0.Next := TRUE;
						idx := idx + 1;
						em.substate := 10;
					ELSE
						idx := 0;
						em.cmd.sc := TRUE;
					END_IF
			END_CASE

		STATE_STARTING:
			CASE em.substate OF
				0:
					em.description := 'start shuttle movement';
					IF MC_BR_SecGetShuttle_AcpTrak_0.TotalCount > 0 THEN
						MC_BR_ElasticMoveVel_AcpTrak_0.Axis 	:= ADR(this.axis[idx]);
						MC_BR_ElasticMoveVel_AcpTrak_0.Execute 	:= TRUE;
						em.substate := 10;
					ELSE
						em.cmd.sc := TRUE; // no shuttles
					END_IF
				10:
					em.description := 'need a scan before checking if the fub is active or in velocity'; //when changing axis (still active from last execute)
					IF MC_BR_ElasticMoveVel_AcpTrak_0.Active THEN
						MC_BR_ElasticMoveVel_AcpTrak_0.Execute := FALSE;
						idx := idx+1;
						em.substate := 20;
					ELSIF MC_BR_ElasticMoveVel_AcpTrak_0.Error THEN
						//todo: error handling
					END_IF
				20:
					em.description := 'move on or next shuttle';
					IF MC_BR_SecGetShuttle_AcpTrak_0.TotalCount = idx THEN
						idx := 0; 	//done
						em.cmd.sc := TRUE;
					ELSE			//next
						em.substate := 0;
					END_IF
			END_CASE

		STATE_EXECUTE:
			em.cmd.sc := TRUE;
			CASE em.substate OF
				0:
					em.description := 'waiting for shuttle';
					IF MC_BR_TrgPointEnable_AcpTrak_0.EventCount > 0 AND MC_BR_TrgPointEnable_AcpTrak_0.Valid THEN
						em.substate := 10;
					END_IF
				10:
					em.description := 'get axis id';
					MC_BR_TrgPointGetInfo_AcpTrak_0.Execute := TRUE;
					IF MC_BR_TrgPointGetInfo_AcpTrak_0.Done THEN
						axis := MC_BR_TrgPointGetInfo_AcpTrak_0.TrgPointInfo.Axis;
						MC_BR_TrgPointGetInfo_AcpTrak_0.Execute := FALSE;
						em.substate := 20;
					END_IF
				20:
					em.description := 'read axis user data';
					MC_BR_ShCopyUserData_AcpTrak_0.Axis 		:= ADR(axis);    				//Zuweisen der Achsreferenz
		            MC_BR_ShCopyUserData_AcpTrak_0.DataAddress 	:= ADR(this.userData);          //Zuweisen der zu lesenden Prozessvariable
		            MC_BR_ShCopyUserData_AcpTrak_0.DataSize 	:= SIZEOF(this.userData);       //Zuweisen der Länge der Prozessvariable
		            MC_BR_ShCopyUserData_AcpTrak_0.Mode 		:= mcACPTRAK_USERDATA_GET;      //Modus auf Schreiben setzen
		            MC_BR_ShCopyUserData_AcpTrak_0.Execute 		:= TRUE;                        //Werte der Prozessvariable auf die Anwenderdaten des Shuttles kopieren
		            IF MC_BR_ShCopyUserData_AcpTrak_0.Done THEN                            		//Kopieren der Werte war erfolgreich
		                MC_BR_ShCopyUserData_AcpTrak_0.Execute := FALSE;
		                em.substate := 30;
		            END_IF
		        30:
					em.description := 'write axis user data';
					MC_BR_ShCopyUserData_AcpTrak_0.Axis 		:= ADR(axis);    				 //Zuweisen der Achsreferenz
					MC_BR_ShCopyUserData_AcpTrak_0.DataAddress 	:= ADR(this.userData);           //Zuweisen der zu beschreibenden Prozessvariable
		            MC_BR_ShCopyUserData_AcpTrak_0.DataSize 	:= SIZEOF(this.userData);        //Zuweisen der Länge der Prozessvariable
		            MC_BR_ShCopyUserData_AcpTrak_0.Mode 		:= mcACPTRAK_USERDATA_SET;       //Modus auf Lesen setzen
		            MC_BR_ShCopyUserData_AcpTrak_0.Execute 		:= TRUE;                         //Werte der Anwenderdaten des Shuttles auf die Prozessvariable kopieren
		            IF MC_BR_ShCopyUserData_AcpTrak_0.Done THEN                            		 //Kopieren der Werte war erfolgreich
		                MC_BR_ShCopyUserData_AcpTrak_0.Execute := FALSE;
		                em.substate := 40;
		            END_IF
				40:
					em.description := 'send shuttle to next sector';
					MC_BR_RoutedMoveVel_AcpTrak_0.Axis 		:= ADR(axis);
					MC_BR_RoutedMoveVel_AcpTrak_0.Execute 	:= TRUE;
					em.substate := 50;
				50:
					em.description := 'need a scan before checking if the fub is active'; //when changing axis
					IF MC_BR_RoutedMoveVel_AcpTrak_0.Active THEN
						MC_BR_RoutedMoveVel_AcpTrak_0.Execute := FALSE;
						em.substate := 0;
					END_IF
			END_CASE

			STATE_CLEARING:
				brsmemset(ADR(this.axis),0,SIZEOF(this.axis));
				em.cmd.sc := TRUE;
	ELSE
		em.cmd.sc := TRUE;
	END_CASE

	em();

	MC_BR_SecGetShuttle_AcpTrak_0();
	MC_BR_TrgPointEnable_AcpTrak_0();
	MC_BR_TrgPointGetInfo_AcpTrak_0();
	MC_BR_RoutedMoveVel_AcpTrak_0();
	MC_BR_ElasticMoveVel_AcpTrak_0();
	MC_BR_ShCopyUserData_AcpTrak_0();
	MC_BR_BarrierCommand_AcpTrak_0();
	IF MC_BR_BarrierCommand_AcpTrak_0.Done THEN
		MC_BR_BarrierCommand_AcpTrak_0.Execute := FALSE;
	END_IF

	MC_BR_BarrierReadInfo_AcpTrak_0(Enable := TRUE);

END_PROGRAM

PROGRAM _EXIT
	(* Insert code here *)

END_PROGRAM
```

#### setup.st
```iecst
ACTION setup:

	gTrack1.velocity     := SEL(gTrack1.velocity <> 0.0, 0.5, gTrack1.velocity); //default 0.5
    gTrack1.acceleration := SEL(gTrack1.acceleration <> 0.0, 1.0, gTrack1.acceleration); //default 1.0
    gTrack1.deceleration := SEL(gTrack1.deceleration <> 0.0, 1.0, gTrack1.deceleration); //default 1.0

	MC_BR_SecGetShuttle_AcpTrak_0.Sector := ADR(SectorTrack1);	//current sector

	MC_BR_TrgPointEnable_AcpTrak_0.Enable := FALSE; //<--- only valid for Track1 (not used)
	MC_BR_TrgPointEnable_AcpTrak_0.ProcessPoint := ADR(PP_Track1);
	MC_BR_TrgPointGetInfo_AcpTrak_0.ProcessPoint := ADR(PP_Track1);

	MC_BR_RoutedMoveVel_AcpTrak_0.Sector 	:= ADR(SectorTrack4); //next sector
	MC_BR_RoutedMoveVel_AcpTrak_0.Position 	:= 0.0;
	MC_BR_RoutedMoveVel_AcpTrak_0.AdvancedParameters.StartDirection 	:= mcDIR_UNDEFINED;
	MC_BR_RoutedMoveVel_AcpTrak_0.AdvancedParameters.EndDirection 		:= mcDIR_UNDEFINED;
	MC_BR_RoutedMoveVel_AcpTrak_0.AdvancedParameters.ShuttleOrientation := mcDIR_UNDEFINED;
	MC_BR_RoutedMoveVel_AcpTrak_0.Velocity 		:= gTrack1.velocity;
	MC_BR_RoutedMoveVel_AcpTrak_0.RouteVelocity := gTrack1.velocity;
	MC_BR_RoutedMoveVel_AcpTrak_0.Acceleration 	:= gTrack1.acceleration;
	MC_BR_RoutedMoveVel_AcpTrak_0.Deceleration 	:= gTrack1.deceleration;

	MC_BR_ElasticMoveVel_AcpTrak_0.Acceleration := gTrack1.acceleration;
	MC_BR_ElasticMoveVel_AcpTrak_0.Deceleration := gTrack1.deceleration;
	MC_BR_ElasticMoveVel_AcpTrak_0.Velocity 	:= gTrack1.velocity;
	MC_BR_ElasticMoveVel_AcpTrak_0.Direction 	:= myTestDirection;

	MC_BR_BarrierCommand_AcpTrak_0.ProcessPoint := ADR(PP_Track1);
	MC_BR_BarrierReadInfo_AcpTrak_0.ProcessPoint := ADR(PP_Track1);

	this.userData.Color := SHUTTLE_COLOR_BLUE;

END_ACTION
```

#### Variables.var - Local variables
```iecst
VAR
	idx : USINT;
	em : brdkEM; (*Equipment module*)
	this : this_typ;
	MC_BR_TrgPointEnable_AcpTrak_0 : MC_BR_TrgPointEnable_AcpTrak;
	MC_BR_TrgPointGetInfo_AcpTrak_0 : MC_BR_TrgPointGetInfo_AcpTrak;
	MC_BR_RoutedMoveVel_AcpTrak_0 : MC_BR_RoutedMoveVel_AcpTrak;
	MC_BR_SecGetShuttle_AcpTrak_0 : MC_BR_SecGetShuttle_AcpTrak;
	MC_BR_ElasticMoveVel_AcpTrak_0 : MC_BR_ElasticMoveVel_AcpTrak;
	axis : McAxisType;
	MC_BR_ShCopyUserData_AcpTrak_0 : MC_BR_ShCopyUserData_AcpTrak;
	MC_BR_BarrierCommand_AcpTrak_0 : MC_BR_BarrierCommand_AcpTrak;
END_VAR
(*Insert your comment here.*)
VAR
	cm : brdkCM;
	MC_BR_TrgPointEnable_PreTrak : MC_BR_TrgPointEnable_AcpTrak;
	MC_BR_TrgPointGetInfo_PreTrak : MC_BR_TrgPointGetInfo_AcpTrak;
	MC_BR_RoutedMoveVel_PreTrak : MC_BR_RoutedMoveVel_AcpTrak;
	MC_BR_BarrierReadInfo_AcpTrak_0 : MC_BR_BarrierReadInfo_AcpTrak;
	myTestDirection : McDirectionEnum;
END_VAR
```

#### Types.typ - Local data types
```iecst
TYPE
	this_typ : 	STRUCT
		axis : ARRAY[0..29]OF McAxisType;
		shiftSector : BOOL;
		userData : ShuttleUserData_typ;
		selector : trak_parameter_selector_typ;
		preAxis : McAxisType;
		counter : USINT;
	END_STRUCT;
END_TYPE
```

### Track1Global.typ - Global data types
```iecst
TYPE
	trak_parameter_typ : 	STRUCT
		velocity : REAL;
		acceleration : REAL;
		deceleration : REAL;
		selector : trak_parameter_selector_typ;
	END_STRUCT;
	trak_parameter_selector_typ :
		(
		TRAK_SELECTOR_ALL := 0,
		TRAK_SELECTOR_NONE := 1,
		TRAK_SELECTOR_2ND := 2,
		TRAK_SELECTOR_3RD := 3,
		TRAK_SELECTOR_4TH := 4
		);
END_TYPE
```

### Track1Global.var - Global variables
```iecst
VAR RETAIN
	gTrack1 : trak_parameter_typ;
END_VAR
```

### Program Logical/Modules/Sectors/Track2Sector/Track2Sector (IEC) - Task for handling Track 2 sectors

- Main.st (reference to Logical/Modules/Sectors/Track1Sector/Track1Sector/Main.st)

#### setup.st
```iecst
ACTION setup:

	gTrack2.velocity     := SEL(gTrack2.velocity <> 0.0, 0.5, gTrack2.velocity); //default 0.5
    gTrack2.acceleration := SEL(gTrack2.acceleration <> 0.0, 1.0, gTrack2.acceleration); //default 1.0
    gTrack2.deceleration := SEL(gTrack2.deceleration <> 0.0, 1.0, gTrack2.deceleration); //default 1.0

	MC_BR_SecGetShuttle_AcpTrak_0.Sector := ADR(SectorTrack2);	//current sector

	MC_BR_TrgPointEnable_AcpTrak_0.ProcessPoint := ADR(PP_Track2);
	MC_BR_TrgPointGetInfo_AcpTrak_0.ProcessPoint := ADR(PP_Track2);

	MC_BR_RoutedMoveVel_AcpTrak_0.Sector 	:= ADR(SectorTrack1); //next sector
	MC_BR_RoutedMoveVel_AcpTrak_0.Position 	:= 0.0;
	MC_BR_RoutedMoveVel_AcpTrak_0.AdvancedParameters.StartDirection 	:= mcDIR_UNDEFINED;
	MC_BR_RoutedMoveVel_AcpTrak_0.AdvancedParameters.EndDirection 		:= mcDIR_POSITIVE;
	MC_BR_RoutedMoveVel_AcpTrak_0.AdvancedParameters.ShuttleOrientation := mcDIR_UNDEFINED;
	MC_BR_RoutedMoveVel_AcpTrak_0.Velocity 		:= gTrack2.velocity;
	MC_BR_RoutedMoveVel_AcpTrak_0.RouteVelocity := gTrack2.velocity;
	MC_BR_RoutedMoveVel_AcpTrak_0.Acceleration 	:= gTrack2.acceleration;
	MC_BR_RoutedMoveVel_AcpTrak_0.Deceleration 	:= gTrack2.deceleration;

	MC_BR_ElasticMoveVel_AcpTrak_0.Acceleration := gTrack2.acceleration;
	MC_BR_ElasticMoveVel_AcpTrak_0.Deceleration := gTrack2.deceleration;
	MC_BR_ElasticMoveVel_AcpTrak_0.Velocity 	:= gTrack2.velocity;
	MC_BR_ElasticMoveVel_AcpTrak_0.Direction 	:= mcDIR_NEGATIVE;

	MC_BR_BarrierCommand_AcpTrak_0.ProcessPoint := ADR(PP_Track2);
	MC_BR_BarrierReadInfo_AcpTrak_0.ProcessPoint := ADR(PP_Track2);

	this.userData.Color := SHUTTLE_COLOR_GREEN;

	//selector pre track
	MC_BR_TrgPointEnable_PreTrak.ProcessPoint := ADR(PP_Pre_Track2);

	MC_BR_TrgPointGetInfo_PreTrak.ProcessPoint := ADR(PP_Pre_Track2);

	MC_BR_RoutedMoveVel_PreTrak.Axis 			:= ADR(this.preAxis);
	MC_BR_RoutedMoveVel_PreTrak.Sector 			:= ADR(SectorTrack2); //this sector
	MC_BR_RoutedMoveVel_PreTrak.Acceleration 	:= gTrack1.acceleration;
	MC_BR_RoutedMoveVel_PreTrak.Deceleration 	:= gTrack1.deceleration;
	MC_BR_RoutedMoveVel_PreTrak.Position	  	:= 0.0;
	MC_BR_RoutedMoveVel_PreTrak.Velocity     	:= gTrack1.velocity;
	MC_BR_RoutedMoveVel_PreTrak.AdvancedParameters.StartDirection 		:= mcDIR_UNDEFINED;
	MC_BR_RoutedMoveVel_PreTrak.AdvancedParameters.EndDirection			:= mcDIR_UNDEFINED;
	MC_BR_RoutedMoveVel_PreTrak.AdvancedParameters.ShuttleOrientation 	:= mcDIR_UNDEFINED;

	this.selector := gTrack2.selector;

	selector;

END_ACTION
```

- Variables.var (reference to Logical/Modules/Sectors/Track1Sector/Track1Sector/Variables.var)

- Types.typ (reference to Logical/Modules/Sectors/Track1Sector/Track1Sector/Types.typ)

#### selector.st
```iecst
ACTION selector:

	CASE cm.state OF
		0:
			MC_BR_TrgPointEnable_PreTrak.Enable := TRUE;
			cm.state := 100;

		100:
			IF MC_BR_TrgPointEnable_PreTrak.EventCount > 0 AND MC_BR_TrgPointEnable_PreTrak.Valid THEN
				MC_BR_TrgPointGetInfo_PreTrak.Execute := TRUE;
				cm.state := 110;
			END_IF

		110:
			IF MC_BR_TrgPointGetInfo_PreTrak.Done THEN
				this.preAxis := MC_BR_TrgPointGetInfo_PreTrak.TrgPointInfo.Axis;
				MC_BR_TrgPointGetInfo_PreTrak.Execute := FALSE;
				cm.state := 120;
			END_IF

		120:
			cm.description := 'evaluate shuttle';
			CASE this.selector OF
				TRAK_SELECTOR_NONE:
					cm.state := 100;

				TRAK_SELECTOR_ALL:
					CASE cm.substate OF
						0:
							MC_BR_RoutedMoveVel_PreTrak.Execute := TRUE;
							cm.substate := 10;
						10:
							IF MC_BR_RoutedMoveVel_PreTrak.Active THEN
								MC_BR_RoutedMoveVel_PreTrak.Execute := FALSE;
								cm.state := 100;
								cm.substate := 0;
							END_IF
					END_CASE

				TRAK_SELECTOR_2ND:
					CASE cm.substate OF
						0:
							IF this.counter >= 1 THEN
								MC_BR_RoutedMoveVel_PreTrak.Execute := TRUE;
								this.counter := 0;
								cm.substate := 10;
							ELSE
								cm.state := 100; // do nothing
								this.counter := this.counter + 1;
							END_IF
						10:
							IF MC_BR_RoutedMoveVel_PreTrak.Active THEN
								MC_BR_RoutedMoveVel_PreTrak.Execute := FALSE;
								cm.state := 100;
								cm.substate := 0;
							END_IF
					END_CASE

				TRAK_SELECTOR_3RD:
					CASE cm.substate OF
						0:
							IF this.counter >= 2 THEN
								MC_BR_RoutedMoveVel_PreTrak.Execute := TRUE;
								this.counter := 0;
								cm.substate := 10;
							ELSE
								cm.state := 100; // do nothing
								this.counter := this.counter + 1;
							END_IF
						10:
							IF MC_BR_RoutedMoveVel_PreTrak.Active THEN
								MC_BR_RoutedMoveVel_PreTrak.Execute := FALSE;
								cm.state := 100;
								cm.substate := 0;
							END_IF
					END_CASE

				TRAK_SELECTOR_4TH:
					CASE cm.substate OF
						0:
							IF this.counter >= 3 THEN
								MC_BR_RoutedMoveVel_PreTrak.Execute := TRUE;
								this.counter := 0;
								cm.substate := 10;
							ELSE
								cm.state := 100; // do nothing
								this.counter := this.counter + 1;
							END_IF
						10:
							IF MC_BR_RoutedMoveVel_PreTrak.Active THEN
								MC_BR_RoutedMoveVel_PreTrak.Execute := FALSE;
								cm.state := 100;
								cm.substate := 0;
							END_IF
					END_CASE
			END_CASE

	END_CASE

	MC_BR_TrgPointEnable_PreTrak();

	MC_BR_TrgPointGetInfo_PreTrak();

	MC_BR_RoutedMoveVel_PreTrak();

	cm();

END_ACTION
```

### Track2Global.var - Global variables
```iecst
VAR RETAIN
	gTrack2 : trak_parameter_typ;
END_VAR
```

### Program Logical/Modules/Sectors/Track3Sector/Track3Sector (IEC)

#### setup.st
```iecst
ACTION setup:

	gTrack3.velocity     := SEL(gTrack3.velocity <> 0.0, 0.5, gTrack3.velocity); //default 0.5
    gTrack3.acceleration := SEL(gTrack3.acceleration <> 0.0, 1.0, gTrack3.acceleration); //default 1.0
    gTrack3.deceleration := SEL(gTrack3.deceleration <> 0.0, 1.0, gTrack3.deceleration); //default 1.0

	MC_BR_SecGetShuttle_AcpTrak_0.Sector := ADR(SectorTrack3);	//current sector

	MC_BR_TrgPointEnable_AcpTrak_0.ProcessPoint := ADR(PP_Track3);
	MC_BR_TrgPointGetInfo_AcpTrak_0.ProcessPoint := ADR(PP_Track3);

	MC_BR_RoutedMoveVel_AcpTrak_0.Sector 	:= ADR(SectorTrack1); //next sector
	MC_BR_RoutedMoveVel_AcpTrak_0.Position 	:= 0.0;
	MC_BR_RoutedMoveVel_AcpTrak_0.AdvancedParameters.StartDirection 	:= mcDIR_UNDEFINED;
	MC_BR_RoutedMoveVel_AcpTrak_0.AdvancedParameters.EndDirection 		:= mcDIR_POSITIVE;
	MC_BR_RoutedMoveVel_AcpTrak_0.AdvancedParameters.ShuttleOrientation := mcDIR_UNDEFINED;
	MC_BR_RoutedMoveVel_AcpTrak_0.Velocity 		:= gTrack3.velocity;
	MC_BR_RoutedMoveVel_AcpTrak_0.RouteVelocity := gTrack3.velocity;
	MC_BR_RoutedMoveVel_AcpTrak_0.Acceleration 	:= gTrack3.acceleration;
	MC_BR_RoutedMoveVel_AcpTrak_0.Deceleration 	:= gTrack3.deceleration;

	MC_BR_ElasticMoveVel_AcpTrak_0.Acceleration := gTrack3.acceleration;
	MC_BR_ElasticMoveVel_AcpTrak_0.Deceleration := gTrack3.deceleration;
	MC_BR_ElasticMoveVel_AcpTrak_0.Velocity 	:= gTrack3.velocity;
	MC_BR_ElasticMoveVel_AcpTrak_0.Direction 	:= mcDIR_NEGATIVE;

	MC_BR_BarrierCommand_AcpTrak_0.ProcessPoint := ADR(PP_Track3);
	MC_BR_BarrierReadInfo_AcpTrak_0.ProcessPoint := ADR(PP_Track3);

	this.userData.Color := SHUTTLE_COLOR_YELLOW;

	//selector pre track
	MC_BR_TrgPointEnable_PreTrak.ProcessPoint := ADR(PP_Pre_Track3);

	MC_BR_TrgPointGetInfo_PreTrak.ProcessPoint := ADR(PP_Pre_Track3);

	MC_BR_RoutedMoveVel_PreTrak.Axis 			:= ADR(this.preAxis);
	MC_BR_RoutedMoveVel_PreTrak.Sector 			:= ADR(SectorTrack3); //this sector
	MC_BR_RoutedMoveVel_PreTrak.Acceleration 	:= gTrack1.acceleration;
	MC_BR_RoutedMoveVel_PreTrak.Deceleration 	:= gTrack1.deceleration;
	MC_BR_RoutedMoveVel_PreTrak.Position	  	:= 0.0;
	MC_BR_RoutedMoveVel_PreTrak.Velocity     	:= gTrack1.velocity;
	MC_BR_RoutedMoveVel_PreTrak.AdvancedParameters.StartDirection 		:= mcDIR_UNDEFINED;
	MC_BR_RoutedMoveVel_PreTrak.AdvancedParameters.EndDirection			:= mcDIR_UNDEFINED;
	MC_BR_RoutedMoveVel_PreTrak.AdvancedParameters.ShuttleOrientation 	:= mcDIR_UNDEFINED;

	this.selector := gTrack3.selector;

	selector;

END_ACTION
```

### Track3Global.var - Global variables
```iecst
VAR RETAIN
	gTrack3 : trak_parameter_typ;
END_VAR
```

### Program Logical/Modules/Sectors/Track4Sector/Track4Sector (IEC)

- Main.st (reference to Logical/Modules/Sectors/Track1Sector/Track1Sector/Main.st)

#### setup.st
```iecst
ACTION setup:

	gTrack4.velocity     := SEL(gTrack4.velocity <> 0.0, 0.5, gTrack4.velocity); //default 0.5
    gTrack4.acceleration := SEL(gTrack4.acceleration <> 0.0, 1.0, gTrack4.acceleration); //default 1.0
    gTrack4.deceleration := SEL(gTrack4.deceleration <> 0.0, 1.0, gTrack4.deceleration); //default 1.0

	MC_BR_SecGetShuttle_AcpTrak_0.Sector := ADR(SectorTrack4);	//current sector

	MC_BR_TrgPointEnable_AcpTrak_0.ProcessPoint := ADR(PP_Track4);
	MC_BR_TrgPointGetInfo_AcpTrak_0.ProcessPoint := ADR(PP_Track4);

	MC_BR_RoutedMoveVel_AcpTrak_0.Sector 	:= ADR(SectorTrack1); //next sector
	MC_BR_RoutedMoveVel_AcpTrak_0.Position 	:= 0.0;
	MC_BR_RoutedMoveVel_AcpTrak_0.AdvancedParameters.StartDirection 	:= mcDIR_UNDEFINED;
	MC_BR_RoutedMoveVel_AcpTrak_0.AdvancedParameters.EndDirection 		:= mcDIR_POSITIVE;
	MC_BR_RoutedMoveVel_AcpTrak_0.AdvancedParameters.ShuttleOrientation := mcDIR_UNDEFINED;
	MC_BR_RoutedMoveVel_AcpTrak_0.Velocity 		:= gTrack4.velocity;
	MC_BR_RoutedMoveVel_AcpTrak_0.RouteVelocity := gTrack4.velocity;
	MC_BR_RoutedMoveVel_AcpTrak_0.Acceleration 	:= gTrack4.acceleration;
	MC_BR_RoutedMoveVel_AcpTrak_0.Deceleration 	:= gTrack4.deceleration;

	MC_BR_ElasticMoveVel_AcpTrak_0.Acceleration := gTrack4.acceleration;
	MC_BR_ElasticMoveVel_AcpTrak_0.Deceleration := gTrack4.deceleration;
	MC_BR_ElasticMoveVel_AcpTrak_0.Velocity 	:= gTrack4.velocity;
	MC_BR_ElasticMoveVel_AcpTrak_0.Direction 	:= mcDIR_NEGATIVE;

	MC_BR_BarrierCommand_AcpTrak_0.ProcessPoint := ADR(PP_Track4);
	MC_BR_BarrierReadInfo_AcpTrak_0.ProcessPoint := ADR(PP_Track4);

	this.userData.Color := SHUTTLE_COLOR_RED;

	//selector pre track
	MC_BR_TrgPointEnable_PreTrak.ProcessPoint := ADR(PP_Pre_Track4);

	MC_BR_TrgPointGetInfo_PreTrak.ProcessPoint := ADR(PP_Pre_Track4);

	MC_BR_RoutedMoveVel_PreTrak.Axis 			:= ADR(this.preAxis);
	MC_BR_RoutedMoveVel_PreTrak.Sector 			:= ADR(SectorTrack4); //this sector
	MC_BR_RoutedMoveVel_PreTrak.Acceleration 	:= gTrack1.acceleration;
	MC_BR_RoutedMoveVel_PreTrak.Deceleration 	:= gTrack1.deceleration;
	MC_BR_RoutedMoveVel_PreTrak.Position	  	:= 0.0;
	MC_BR_RoutedMoveVel_PreTrak.Velocity     	:= gTrack1.velocity;
	MC_BR_RoutedMoveVel_PreTrak.AdvancedParameters.StartDirection 		:= mcDIR_UNDEFINED;
	MC_BR_RoutedMoveVel_PreTrak.AdvancedParameters.EndDirection			:= mcDIR_UNDEFINED;
	MC_BR_RoutedMoveVel_PreTrak.AdvancedParameters.ShuttleOrientation 	:= mcDIR_UNDEFINED;

	this.selector := gTrack4.selector;

	selector;

END_ACTION
```

- Variables.var (reference to Logical/Modules/Sectors/Track1Sector/Track1Sector/Variables.var)

- Types.typ (reference to Logical/Modules/Sectors/Track1Sector/Track1Sector/Types.typ)

- selector.st (reference to Logical/Modules/Sectors/Track2Sector/Track2Sector/selector.st)

### Track4Global.var - Global variables
```iecst
VAR RETAIN
	gTrack4 : trak_parameter_typ;
END_VAR
```

### Program Logical/Modules/Sectors/Track5Sector/Track5Sector (IEC)

#### setup.st
```iecst
ACTION setup:

	gTrack5.velocity     := SEL(gTrack5.velocity <> 0.0, 0.5, gTrack5.velocity); //default 0.5
    gTrack5.acceleration := SEL(gTrack5.acceleration <> 0.0, 1.0, gTrack5.acceleration); //default 1.0
    gTrack5.deceleration := SEL(gTrack5.deceleration <> 0.0, 1.0, gTrack5.deceleration); //default 1.0

	MC_BR_SecGetShuttle_AcpTrak_0.Sector := ADR(SectorTrack5);	//current sector

	MC_BR_TrgPointEnable_AcpTrak_0.ProcessPoint := ADR(PP_Track5);
	MC_BR_TrgPointGetInfo_AcpTrak_0.ProcessPoint := ADR(PP_Track5);

	MC_BR_RoutedMoveVel_AcpTrak_0.Sector 	:= ADR(SectorTrack1); //next sector
	MC_BR_RoutedMoveVel_AcpTrak_0.Position 	:= 0.0;
	MC_BR_RoutedMoveVel_AcpTrak_0.AdvancedParameters.StartDirection 	:= mcDIR_POSITIVE;
	MC_BR_RoutedMoveVel_AcpTrak_0.AdvancedParameters.EndDirection 		:= mcDIR_NEGATIVE;
	MC_BR_RoutedMoveVel_AcpTrak_0.AdvancedParameters.ShuttleOrientation := mcDIR_NEGATIVE;
	MC_BR_RoutedMoveVel_AcpTrak_0.Velocity 		:= gTrack5.velocity;
	MC_BR_RoutedMoveVel_AcpTrak_0.RouteVelocity := gTrack5.velocity;
	MC_BR_RoutedMoveVel_AcpTrak_0.Acceleration 	:= gTrack5.acceleration;
	MC_BR_RoutedMoveVel_AcpTrak_0.Deceleration 	:= gTrack5.deceleration;

	MC_BR_ElasticMoveVel_AcpTrak_0.Acceleration := gTrack5.acceleration;
	MC_BR_ElasticMoveVel_AcpTrak_0.Deceleration := gTrack5.deceleration;
	MC_BR_ElasticMoveVel_AcpTrak_0.Velocity 	:= gTrack5.velocity;
	MC_BR_ElasticMoveVel_AcpTrak_0.Direction 	:= mcDIR_POSITIVE;

	MC_BR_BarrierCommand_AcpTrak_0.ProcessPoint := ADR(PP_Track5);
	MC_BR_BarrierReadInfo_AcpTrak_0.ProcessPoint := ADR(PP_Track5);

	this.userData.Color := SHUTTLE_COLOR_CYAN;

END_ACTION
```

### Track5Global.var - Global variables
```iecst
VAR RETAIN
	gTrack5 : trak_parameter_typ;
END_VAR
```

### Program Logical/Modules/Sectors/Track6Sector/Track6Sector (IEC)

- Main.st (reference to Logical/Modules/Sectors/Track1Sector/Track1Sector/Main.st)

#### setup.st
```iecst
ACTION setup:

	gTrack6.velocity     := SEL(gTrack6.velocity <> 0.0, 0.5, gTrack6.velocity); //default 0.5
    gTrack6.acceleration := SEL(gTrack6.acceleration <> 0.0, 1.0, gTrack6.acceleration); //default 1.0
    gTrack6.deceleration := SEL(gTrack6.deceleration <> 0.0, 1.0, gTrack6.deceleration); //default 1.0

	MC_BR_SecGetShuttle_AcpTrak_0.Sector := ADR(SectorTrack6);	//current sector

	MC_BR_TrgPointEnable_AcpTrak_0.ProcessPoint := ADR(PP_Track6);
	MC_BR_TrgPointGetInfo_AcpTrak_0.ProcessPoint := ADR(PP_Track6);

	MC_BR_RoutedMoveVel_AcpTrak_0.Sector 	:= ADR(SectorTrack1); //next sector
	MC_BR_RoutedMoveVel_AcpTrak_0.Position 	:= 3.0;
	MC_BR_RoutedMoveVel_AcpTrak_0.AdvancedParameters.StartDirection 	:= mcDIR_UNDEFINED;
	MC_BR_RoutedMoveVel_AcpTrak_0.AdvancedParameters.EndDirection 		:= mcDIR_POSITIVE;
	MC_BR_RoutedMoveVel_AcpTrak_0.AdvancedParameters.ShuttleOrientation := mcDIR_UNDEFINED;
	MC_BR_RoutedMoveVel_AcpTrak_0.Velocity 		:= gTrack6.velocity;
	MC_BR_RoutedMoveVel_AcpTrak_0.RouteVelocity := gTrack6.velocity;
	MC_BR_RoutedMoveVel_AcpTrak_0.Acceleration 	:= gTrack6.acceleration;
	MC_BR_RoutedMoveVel_AcpTrak_0.Deceleration 	:= gTrack6.deceleration;

	MC_BR_ElasticMoveVel_AcpTrak_0.Acceleration := gTrack6.acceleration;
	MC_BR_ElasticMoveVel_AcpTrak_0.Deceleration := gTrack6.deceleration;
	MC_BR_ElasticMoveVel_AcpTrak_0.Velocity 	:= gTrack6.velocity;
	MC_BR_ElasticMoveVel_AcpTrak_0.Direction 	:= mcDIR_POSITIVE;

	MC_BR_BarrierCommand_AcpTrak_0.ProcessPoint := ADR(PP_Track6);
	MC_BR_BarrierReadInfo_AcpTrak_0.ProcessPoint := ADR(PP_Track6);

	this.userData.Color := SHUTTLE_COLOR_ORANGE;

END_ACTION
```

- Types.typ (reference to Logical/Modules/Sectors/Track1Sector/Track1Sector/Types.typ)

- Variables.var (reference to Logical/Modules/Sectors/Track1Sector/Track1Sector/Variables.var)

### Track6Global.var - Global variables
```iecst
VAR RETAIN
	gTrack6 : trak_parameter_typ;
END_VAR
```

### Package Logical/Modules/Safety - Safety interface task

### Program Logical/Modules/Safety/Safety (IEC)

#### Types.typ
```iecst
TYPE
	safety_typ : 	STRUCT
		cmd : safety_cmd_typ;
		status : safety_status_typ;
	END_STRUCT;
	safety_cmd_typ : 	STRUCT
		reset : BOOL; (*command for resetting safety*)
	END_STRUCT;
	safety_status_typ : 	STRUCT
		safetyStarted : BOOL; (*TRUE if safety application is running*)
		safetyOk : BOOL; (*TRUE if safety chain ok and reset not needed*)
		resetNeeded : BOOL; (*TRUE if safety has tripped and needs a reset*)
	END_STRUCT;
END_TYPE
```

#### Variables.var
```iecst
VAR
	this : safety_typ; (*local struct*)
END_VAR
```

#### Main.st
```iecst
PROGRAM _INIT
	(* Insert code here *)
	 this;
END_PROGRAM

PROGRAM _CYCLIC
	(* Insert code here *)

END_PROGRAM

PROGRAM _EXIT
	(* Insert code here *)

END_PROGRAM
```

### Program Logical/Simulation/Simulation (IEC)

#### Variables.var
```iecst
VAR
Vis : McAcpTrakAssemblyVisData;
    SizeofVis : UDINT := 0;
    NumVisShuttle : USINT := 0;
    i : USINT := 0;
    pUserData : REFERENCE TO ShuttleUserData_typ;
END_VAR
```

#### Main.st
```iecst
PROGRAM _INIT

    // size of Vis structure - this value has to be entered in B&R scene viewer (PVI -> Options -> Size)
	SizeofVis := SIZEOF(Vis);
	// max number of displayed shuttles
	NumVisShuttle := SIZEOF(Vis.Shuttle) / SIZEOF(Vis.Shuttle[0]);

END_PROGRAM

PROGRAM _CYCLIC

	FOR i:=0 TO (NumVisShuttle-1) DO
		IF gShuttleMon.Shuttle[i].Available THEN
			// format selected monitor data to fit B&R scene viewer
			Vis.Shuttle[i].Available    	:= 1;
			Vis.Shuttle[i].PositionX    	:= LREAL_TO_REAL(gShuttleMon.Shuttle[i].Position.X);
			Vis.Shuttle[i].PositionY    	:= LREAL_TO_REAL(gShuttleMon.Shuttle[i].Position.Y);
			Vis.Shuttle[i].RotationZ    	:= LREAL_TO_REAL(gShuttleMon.Shuttle[i].Orientation.Angle1);
			Vis.Shuttle[i].ExtentToFront    := LREAL_TO_REAL(gShuttleMon.Shuttle[i].ExtentToFront);
			Vis.Shuttle[i].ExtentToBack     := LREAL_TO_REAL(gShuttleMon.Shuttle[i].ExtentToBack);
			Vis.Shuttle[i].Width    		:= LREAL_TO_REAL(gShuttleMon.Shuttle[i].Width);
			brsitoa(gShuttleMon.Shuttle[i].Index, ADR(Vis.Shuttle[i].Text));
			// example: set shuttle colour via user data
			IF gShuttleMon.Shuttle[i].UserData <> 0 THEN
				pUserData ACCESS gShuttleMon.Shuttle[i].UserData;    // access to user data of this shuttle
				IF pUserData.Color = SHUTTLE_COLOR_GREEN THEN
					Vis.Shuttle[i].ColorRed    := 0.0;
					Vis.Shuttle[i].ColorGreen  := 1.0;
					Vis.Shuttle[i].ColorBlue   := 0.0;
				ELSIF pUserData.Color = SHUTTLE_COLOR_BLUE THEN
					Vis.Shuttle[i].ColorRed    := 0.0;
					Vis.Shuttle[i].ColorGreen  := 0.0;
					Vis.Shuttle[i].ColorBlue   := 1.0;
				ELSIF pUserData.Color = SHUTTLE_COLOR_RED THEN
					Vis.Shuttle[i].ColorRed		:= 1.0;
					Vis.Shuttle[i].ColorGreen	:= 0.0;
					Vis.Shuttle[i].ColorBlue	:= 0.0;
				ELSIF pUserData.Color = SHUTTLE_COLOR_ORANGE THEN
					Vis.Shuttle[i].ColorRed		:= 1.0;
					Vis.Shuttle[i].ColorGreen	:= 0.5;
					Vis.Shuttle[i].ColorBlue	:= 0.0;
				ELSIF pUserData.Color = SHUTTLE_COLOR_GREY THEN
					Vis.Shuttle[i].ColorRed		:= 0.75;
					Vis.Shuttle[i].ColorGreen	:= 0.75;
					Vis.Shuttle[i].ColorBlue	:= 0.75;
				ELSIF pUserData.Color = SHUTTLE_COLOR_WHITE THEN
					Vis.Shuttle[i].ColorRed		:= 1.0;
					Vis.Shuttle[i].ColorGreen	:= 1.0;
					Vis.Shuttle[i].ColorBlue	:= 1.0;
				ELSIF pUserData.Color = SHUTTLE_COLOR_BLACK THEN
					Vis.Shuttle[i].ColorRed		:= 0.0;
					Vis.Shuttle[i].ColorGreen	:= 0.0;
					Vis.Shuttle[i].ColorBlue	:= 0.0;
				ELSIF pUserData.Color = SHUTTLE_COLOR_CYAN THEN
					Vis.Shuttle[i].ColorRed		:= 0.0;
					Vis.Shuttle[i].ColorGreen	:= 1.0;
					Vis.Shuttle[i].ColorBlue	:= 1.0;
				ELSIF pUserData.Color = SHUTTLE_COLOR_YELLOW THEN
					Vis.Shuttle[i].ColorRed		:= 1.0;
					Vis.Shuttle[i].ColorGreen	:= 1.0;
					Vis.Shuttle[i].ColorBlue	:= 0.0;
				ELSIF pUserData.Color = SHUTTLE_COLOR_BROWN THEN
					Vis.Shuttle[i].ColorRed		:= 0.5;
					Vis.Shuttle[i].ColorGreen	:= 0.25;
					Vis.Shuttle[i].ColorBlue	:= 0.25;
				ELSIF pUserData.Color = SHUTTLE_COLOR_PINK THEN
					Vis.Shuttle[i].ColorRed		:= 1.0;
					Vis.Shuttle[i].ColorGreen	:= 0.0;
					Vis.Shuttle[i].ColorBlue	:= 1.0;
				END_IF
			END_IF

		ELSE
		//	brsmemset(ADR(Vis.Shuttle[i]), 0, SIZEOF(Vis.Shuttle[0]));
		END_IF
	END_FOR

END_PROGRAM

PROGRAM _EXIT
	(* Insert code here *)

END_PROGRAM
```

### SimulationGlobal.typ
```iecst
TYPE
	ShuttleUserData_typ : 	STRUCT
		Color : ShuttleColor_enum; (*example: product colour*)
		Weight : REAL; (*example: product weight*)
		Partnumber : UDINT; (*example: product part number*)
	END_STRUCT;
	ShuttleColor_enum :
		(
		SHUTTLE_COLOR_GREY := 0,
		SHUTTLE_COLOR_GREEN := 1,
		SHUTTLE_COLOR_RED := 2,
		SHUTTLE_COLOR_BLUE := 3,
		SHUTTLE_COLOR_WHITE := 4,
		SHUTTLE_COLOR_BLACK := 5,
		SHUTTLE_COLOR_YELLOW := 6,
		SHUTTLE_COLOR_PINK := 7,
		SHUTTLE_COLOR_BROWN := 8,
		SHUTTLE_COLOR_CYAN := 9,
		SHUTTLE_COLOR_ORANGE := 10
		);
END_TYPE
```

### Program Logical/Services/Alarm/Alarm (IEC)

#### Variables.var
```iecst
VAR
	MpAlarmXCore_0 : MpAlarmXCore;
	MpAlarmXHistory_0 : MpAlarmXHistory;
END_VAR
```

#### Main.st
```iecst
PROGRAM _INIT

	MpAlarmXCore_0(MpLink:=ADR(gAlarmXCore), Enable:=TRUE);

	MpAlarmXHistory_0(MpLink:=ADR(gAlarmXHistory), Enable:=TRUE);

END_PROGRAM

PROGRAM _CYCLIC

	MpAlarmXCore_0(MpLink:=ADR(gAlarmXCore));

	MpAlarmXHistory_0(MpLink:=ADR(gAlarmXHistory));

END_PROGRAM

PROGRAM _EXIT
	(* Insert code here *)

END_PROGRAM
```

- Visualisation Logical/mappView (not shown)

Listed in the project but not available here: Logical/Global.typ, Logical/Libraries/brdkMU/brdkMU.typ, Logical/Libraries/brdkMU/brdkCM.typ, Logical/Libraries/brdkMU/brdkUM.typ, Logical/Libraries/brdkMU/brdkEMStateToA.c, Logical/Libraries/brdkMU/brdkEMSleep.c, Logical/Libraries/brdkMU/brdkEM_func.h, Logical/Libraries/brdkMU/brdkCM.c, Logical/Libraries/brdkMU/brdkCMChangeParent.c, Logical/Libraries/brdkMU/brdkCMSleep.c, Logical/Libraries/brdkMU/brdkCM_func.h, Logical/Libraries/brdkMU/brdkUM.c, Logical/Libraries/brdkMU/brdkUM_func.h, Logical/Libraries/brdkMU/brdkUM_func.c, Logical/Libraries/brdkMU/brdkMU_func.h, Logical/Libraries/brdkSTR/brdkSTR.typ, Logical/Libraries/brdkSTR/brdkSTR.var, Logical/Libraries/brdkSTR/brdkStrAppendUdintToA.c, Logical/Libraries/brdkSTR/brdkStrAToDint.c, Logical/Libraries/brdkSTR/brdkStrAToUdint.c, Logical/Libraries/brdkSTR/brdkStrCat.c, Logical/Libraries/brdkSTR/brdkStrCatAtChar.c, Logical/Libraries/brdkSTR/brdkStrCharAt.c, Logical/Libraries/brdkSTR/brdkStrCharCount.c, Logical/Libraries/brdkSTR/brdkStrCmp.c, Logical/Libraries/brdkSTR/brdkStrCpy.c, Logical/Libraries/brdkSTR/brdkStrCrc32.c, Logical/Libraries/brdkSTR/brdkStrDintToA.c, Logical/Libraries/brdkSTR/brdkStrEncode.c, Logical/Libraries/brdkSTR/brdkStrFill.c, Logical/Libraries/brdkSTR/brdkStrIndexOf.c, Logical/Libraries/brdkSTR/brdkStrInsertAtPos.c, Logical/Libraries/brdkSTR/brdkStrIsEmpty.c, Logical/Libraries/brdkSTR/brdkStrLen.c, Logical/Libraries/brdkSTR/brdkStrMemCmp.c, Logical/Libraries/brdkSTR/brdkStrMemCpy.c, Logical/Libraries/brdkSTR/brdkStrMemMove.c, Logical/Libraries/brdkSTR/brdkStrMemSet.c, Logical/Libraries/brdkSTR/brdkStrMove.c, Logical/Libraries/brdkSTR/brdkStrNCpy.c, Logical/Libraries/brdkSTR/brdkStrRemove.c, Logical/Libraries/brdkSTR/brdkStrRepeat.c, Logical/Libraries/brdkSTR/brdkStrReplace.c, Logical/Libraries/brdkSTR/brdkStrReverse.c, Logical/Libraries/brdkSTR/brdkStrReverseWords.c, Logical/Libraries/brdkSTR/brdkStrSearch.c, Logical/Libraries/brdkSTR/brdkStrSlice.c, Logical/Libraries/brdkSTR/brdkStrSubStr.c, Logical/Libraries/brdkSTR/brdkStrToDec.c, Logical/Libraries/brdkSTR/brdkStrToHex.c, Logical/Libraries/brdkSTR/brdkStrToLowerCase.c, Logical/Libraries/brdkSTR/brdkStrToUpperCase.c, Logical/Libraries/brdkSTR/brdkStrToUpperCaseWords.c, Logical/Libraries/brdkSTR/brdkStrTrim.c, Logical/Libraries/brdkSTR/brdkStrUdintToA.c, Logical/Libraries/brdkSTR/brdkSTR_func.h, Logical/Libraries/brdkSTR/brdkSTR_func.c, Logical/Simulation/SimulationGlobal.var, Logical/Services/Alarm/AlarmGlobal.typ, Logical/Services/Alarm/AlarmGlobal.var
